(* Logix 5000 project; controller QW361 vendor 1 type 14 code 107 rev 32.11; software revision 32.00; part 16 of 20 *)

        [2374].log_data[1].valid := 1, [2374].log_data[2].valid := 1, [2374].log_data[3].valid := 1, [2374].log_data[4].valid := 1, [2374].time.Year := 2022, [2374].time.Month := 5, [2374].time.Day := 2, [2374].time.Hour := 3, [2374].time.Minute := 24, [2374].time.Second := 59, [2374].time.DST_ON := 1, [2375].log_data[0].min := 1.0, [2375].log_data[0].max := 1.0, [2375].log_data[0].total := 300.0, [2375].log_data[0].time := 300.0, [2375].log_data[0].minminute := 25, [2375].log_data[0].maxminute := 25, [2375].log_data[0].valid := 1, [2375].log_data[1].valid := 1, [2375].log_data[2].valid := 1, [2375].log_data[3].valid := 1, [2375].log_data[4].valid := 1, [2375].time.Year := 2022, [2375].time.Month := 5, [2375].time.Day := 2, [2375].time.Hour := 3, [2375].time.Minute := 29, [2375].time.Second := 59, [2375].time.DST_ON := 1, [2376].log_data[0].min := 1.0, [2376].log_data[0].max := 1.0, [2376].log_data[0].total := 300.0, [2376].log_data[0].time := 300.0, [2376].log_data[0].minminute := 30, [2376].log_data[0].maxminute := 30, [2376].log_data[0].valid := 1, [2376].log_data[1].valid := 1, [2376].log_data[2].valid := 1, [2376].log_data[3].valid := 1, [2376].log_data[4].valid := 1, [2376].time.Year := 2022, [2376].time.Month := 5, [2376].time.Day := 2, [2376].time.Hour := 3, [2376].time.Minute := 34, [2376].time.Second := 59, [2376].time.DST_ON := 1, [2377].log_data[0].min := 1.0, [2377].log_data[0].max := 1.0, [2377].log_data[0].total := 300.0, [2377].log_data[0].time := 300.0, [2377].log_data[0].minminute := 35, [2377].log_data[0].maxminute := 35, [2377].log_data[0].valid := 1, [2377].log_data[1].valid := 1, [2377].log_data[2].valid := 1, [2377].log_data[3].valid := 1, [2377].log_data[4].valid := 1, [2377].time.Year := 2022, [2377].time.Month := 5,
        [2377].time.Day := 2, [2377].time.Hour := 3, [2377].time.Minute := 39, [2377].time.Second := 59, [2377].time.DST_ON := 1, [2378].log_data[0].min := 1.0, [2378].log_data[0].max := 1.0, [2378].log_data[0].total := 300.0, [2378].log_data[0].time := 300.0, [2378].log_data[0].minminute := 40, [2378].log_data[0].maxminute := 40, [2378].log_data[0].valid := 1, [2378].log_data[1].valid := 1, [2378].log_data[2].valid := 1, [2378].log_data[3].valid := 1, [2378].log_data[4].valid := 1, [2378].time.Year := 2022, [2378].time.Month := 5, [2378].time.Day := 2, [2378].time.Hour := 3, [2378].time.Minute := 44, [2378].time.Second := 59, [2378].time.DST_ON := 1, [2379].log_data[0].min := 1.0, [2379].log_data[0].max := 1.0, [2379].log_data[0].total := 300.0, [2379].log_data[0].time := 300.0, [2379].log_data[0].minminute := 45, [2379].log_data[0].maxminute := 45, [2379].log_data[0].valid := 1, [2379].log_data[1].valid := 1, [2379].log_data[2].valid := 1, [2379].log_data[3].valid := 1, [2379].log_data[4].valid := 1, [2379].time.Year := 2022, [2379].time.Month := 5, [2379].time.Day := 2, [2379].time.Hour := 3, [2379].time.Minute := 49, [2379].time.Second := 59, [2379].time.DST_ON := 1, [2380].log_data[0].min := 1.0, [2380].log_data[0].max := 1.0, [2380].log_data[0].total := 300.0, [2380].log_data[0].time := 300.0, [2380].log_data[0].minminute := 50, [2380].log_data[0].maxminute := 50, [2380].log_data[0].valid := 1, [2380].log_data[1].valid := 1, [2380].log_data[2].valid := 1, [2380].log_data[3].valid := 1, [2380].log_data[4].valid := 1, [2380].time.Year := 2022, [2380].time.Month := 5, [2380].time.Day := 2, [2380].time.Hour := 3, [2380].time.Minute := 54, [2380].time.Second := 59, [2380].time.DST_ON := 1, [2381].log_data[0].min := 1.0,
        [2381].log_data[0].max := 1.0, [2381].log_data[0].total := 300.0, [2381].log_data[0].time := 300.0, [2381].log_data[0].minminute := 55, [2381].log_data[0].maxminute := 55, [2381].log_data[0].valid := 1, [2381].log_data[1].valid := 1, [2381].log_data[2].valid := 1, [2381].log_data[3].valid := 1, [2381].log_data[4].valid := 1, [2381].time.Year := 2022, [2381].time.Month := 5, [2381].time.Day := 2, [2381].time.Hour := 3, [2381].time.Minute := 59, [2381].time.Second := 59, [2381].time.DST_ON := 1, [2382].log_data[0].min := 1.0, [2382].log_data[0].max := 1.0, [2382].log_data[0].total := 300.0, [2382].log_data[0].time := 300.0, [2382].log_data[0].valid := 1, [2382].log_data[1].valid := 1, [2382].log_data[2].valid := 1, [2382].log_data[3].valid := 1, [2382].log_data[4].valid := 1, [2382].time.Year := 2022, [2382].time.Month := 5, [2382].time.Day := 2, [2382].time.Hour := 4, [2382].time.Minute := 4, [2382].time.Second := 59, [2382].time.DST_ON := 1, [2383].log_data[0].min := 1.0, [2383].log_data[0].max := 1.0, [2383].log_data[0].total := 300.0, [2383].log_data[0].time := 300.0, [2383].log_data[0].minminute := 5, [2383].log_data[0].maxminute := 5, [2383].log_data[0].valid := 1, [2383].log_data[1].valid := 1, [2383].log_data[2].valid := 1, [2383].log_data[3].valid := 1, [2383].log_data[4].valid := 1, [2383].time.Year := 2022, [2383].time.Month := 5, [2383].time.Day := 2, [2383].time.Hour := 4, [2383].time.Minute := 9, [2383].time.Second := 59, [2383].time.DST_ON := 1, [2384].log_data[0].min := 1.0, [2384].log_data[0].max := 1.0, [2384].log_data[0].total := 300.0, [2384].log_data[0].time := 300.0, [2384].log_data[0].minminute := 10, [2384].log_data[0].maxminute := 10, [2384].log_data[0].valid := 1, [2384].log_data[1].valid := 1, [2384].log_data[2].valid := 1,
        [2384].log_data[3].valid := 1, [2384].log_data[4].valid := 1, [2384].time.Year := 2022, [2384].time.Month := 5, [2384].time.Day := 2, [2384].time.Hour := 4, [2384].time.Minute := 14, [2384].time.Second := 59, [2384].time.DST_ON := 1, [2385].log_data[0].min := 1.0, [2385].log_data[0].max := 1.0, [2385].log_data[0].total := 300.0, [2385].log_data[0].time := 300.0, [2385].log_data[0].minminute := 15, [2385].log_data[0].maxminute := 15, [2385].log_data[0].valid := 1, [2385].log_data[1].valid := 1, [2385].log_data[2].valid := 1, [2385].log_data[3].valid := 1, [2385].log_data[4].valid := 1, [2385].time.Year := 2022, [2385].time.Month := 5, [2385].time.Day := 2, [2385].time.Hour := 4, [2385].time.Minute := 19, [2385].time.Second := 59, [2385].time.DST_ON := 1, [2386].log_data[0].min := 1.0, [2386].log_data[0].max := 1.0, [2386].log_data[0].total := 300.0, [2386].log_data[0].time := 300.0, [2386].log_data[0].minminute := 20, [2386].log_data[0].maxminute := 20, [2386].log_data[0].valid := 1, [2386].log_data[1].valid := 1, [2386].log_data[2].valid := 1, [2386].log_data[3].valid := 1, [2386].log_data[4].valid := 1, [2386].time.Year := 2022, [2386].time.Month := 5, [2386].time.Day := 2, [2386].time.Hour := 4, [2386].time.Minute := 24, [2386].time.Second := 59, [2386].time.DST_ON := 1, [2387].log_data[0].min := 1.0, [2387].log_data[0].max := 1.0, [2387].log_data[0].total := 300.0, [2387].log_data[0].time := 300.0, [2387].log_data[0].minminute := 25, [2387].log_data[0].maxminute := 25, [2387].log_data[0].valid := 1, [2387].log_data[1].valid := 1, [2387].log_data[2].valid := 1, [2387].log_data[3].valid := 1, [2387].log_data[4].valid := 1, [2387].time.Year := 2022, [2387].time.Month := 5, [2387].time.Day := 2, [2387].time.Hour := 4,
        [2387].time.Minute := 29, [2387].time.Second := 59, [2387].time.DST_ON := 1, [2388].log_data[0].min := 1.0, [2388].log_data[0].max := 1.0, [2388].log_data[0].total := 300.0, [2388].log_data[0].time := 300.0, [2388].log_data[0].minminute := 30, [2388].log_data[0].maxminute := 30, [2388].log_data[0].valid := 1, [2388].log_data[1].valid := 1, [2388].log_data[2].valid := 1, [2388].log_data[3].valid := 1, [2388].log_data[4].valid := 1, [2388].time.Year := 2022, [2388].time.Month := 5, [2388].time.Day := 2, [2388].time.Hour := 4, [2388].time.Minute := 34, [2388].time.Second := 59, [2388].time.DST_ON := 1, [2389].log_data[0].min := 1.0, [2389].log_data[0].max := 1.0, [2389].log_data[0].total := 300.0, [2389].log_data[0].time := 300.0, [2389].log_data[0].minminute := 35, [2389].log_data[0].maxminute := 35, [2389].log_data[0].valid := 1, [2389].log_data[1].valid := 1, [2389].log_data[2].valid := 1, [2389].log_data[3].valid := 1, [2389].log_data[4].valid := 1, [2389].time.Year := 2022, [2389].time.Month := 5, [2389].time.Day := 2, [2389].time.Hour := 4, [2389].time.Minute := 39, [2389].time.Second := 59, [2389].time.DST_ON := 1, [2390].log_data[0].min := 1.0, [2390].log_data[0].max := 1.0, [2390].log_data[0].total := 300.0, [2390].log_data[0].time := 300.0, [2390].log_data[0].minminute := 40, [2390].log_data[0].maxminute := 40, [2390].log_data[0].valid := 1, [2390].log_data[1].valid := 1, [2390].log_data[2].valid := 1, [2390].log_data[3].valid := 1, [2390].log_data[4].valid := 1, [2390].time.Year := 2022, [2390].time.Month := 5, [2390].time.Day := 2, [2390].time.Hour := 4, [2390].time.Minute := 44, [2390].time.Second := 59, [2390].time.DST_ON := 1, [2391].log_data[0].min := 1.0, [2391].log_data[0].max := 1.0, [2391].log_data[0].total := 300.0,
        [2391].log_data[0].time := 300.0, [2391].log_data[0].minminute := 45, [2391].log_data[0].maxminute := 45, [2391].log_data[0].valid := 1, [2391].log_data[1].valid := 1, [2391].log_data[2].valid := 1, [2391].log_data[3].valid := 1, [2391].log_data[4].valid := 1, [2391].time.Year := 2022, [2391].time.Month := 5, [2391].time.Day := 2, [2391].time.Hour := 4, [2391].time.Minute := 49, [2391].time.Second := 59, [2391].time.DST_ON := 1, [2392].log_data[0].min := 1.0, [2392].log_data[0].max := 1.0, [2392].log_data[0].total := 300.0, [2392].log_data[0].time := 300.0, [2392].log_data[0].minminute := 50, [2392].log_data[0].maxminute := 50, [2392].log_data[0].valid := 1, [2392].log_data[1].valid := 1, [2392].log_data[2].valid := 1, [2392].log_data[3].valid := 1, [2392].log_data[4].valid := 1, [2392].time.Year := 2022, [2392].time.Month := 5, [2392].time.Day := 2, [2392].time.Hour := 4, [2392].time.Minute := 54, [2392].time.Second := 59, [2392].time.DST_ON := 1, [2393].log_data[0].min := 1.0, [2393].log_data[0].max := 1.0, [2393].log_data[0].total := 300.0, [2393].log_data[0].time := 300.0, [2393].log_data[0].minminute := 55, [2393].log_data[0].maxminute := 55, [2393].log_data[0].valid := 1, [2393].log_data[1].valid := 1, [2393].log_data[2].valid := 1, [2393].log_data[3].valid := 1, [2393].log_data[4].valid := 1, [2393].time.Year := 2022, [2393].time.Month := 5, [2393].time.Day := 2, [2393].time.Hour := 4, [2393].time.Minute := 59, [2393].time.Second := 59, [2393].time.DST_ON := 1, [2394].log_data[0].min := 1.0, [2394].log_data[0].max := 1.0, [2394].log_data[0].total := 300.0, [2394].log_data[0].time := 300.0, [2394].log_data[0].valid := 1, [2394].log_data[1].valid := 1, [2394].log_data[2].valid := 1, [2394].log_data[3].valid := 1, [2394].log_data[4].valid := 1,
        [2394].time.Year := 2022, [2394].time.Month := 5, [2394].time.Day := 2, [2394].time.Hour := 5, [2394].time.Minute := 4, [2394].time.Second := 59, [2394].time.DST_ON := 1, [2395].log_data[0].min := 1.0, [2395].log_data[0].max := 1.0, [2395].log_data[0].total := 300.0, [2395].log_data[0].time := 300.0, [2395].log_data[0].minminute := 5, [2395].log_data[0].maxminute := 5, [2395].log_data[0].valid := 1, [2395].log_data[1].valid := 1, [2395].log_data[2].valid := 1, [2395].log_data[3].valid := 1, [2395].log_data[4].valid := 1, [2395].time.Year := 2022, [2395].time.Month := 5, [2395].time.Day := 2, [2395].time.Hour := 5, [2395].time.Minute := 9, [2395].time.Second := 59, [2395].time.DST_ON := 1, [2396].log_data[0].min := 1.0, [2396].log_data[0].max := 1.0, [2396].log_data[0].total := 300.0, [2396].log_data[0].time := 300.0, [2396].log_data[0].minminute := 10, [2396].log_data[0].maxminute := 10, [2396].log_data[0].valid := 1, [2396].log_data[1].valid := 1, [2396].log_data[2].valid := 1, [2396].log_data[3].valid := 1, [2396].log_data[4].valid := 1, [2396].time.Year := 2022, [2396].time.Month := 5, [2396].time.Day := 2, [2396].time.Hour := 5, [2396].time.Minute := 14, [2396].time.Second := 59, [2396].time.DST_ON := 1, [2397].log_data[0].min := 1.0, [2397].log_data[0].max := 1.0, [2397].log_data[0].total := 300.0, [2397].log_data[0].time := 300.0, [2397].log_data[0].minminute := 15, [2397].log_data[0].maxminute := 15, [2397].log_data[0].valid := 1, [2397].log_data[1].valid := 1, [2397].log_data[2].valid := 1, [2397].log_data[3].valid := 1, [2397].log_data[4].valid := 1, [2397].time.Year := 2022, [2397].time.Month := 5, [2397].time.Day := 2, [2397].time.Hour := 5, [2397].time.Minute := 19, [2397].time.Second := 59,
        [2397].time.DST_ON := 1, [2398].log_data[0].min := 1.0, [2398].log_data[0].max := 1.0, [2398].log_data[0].total := 300.0, [2398].log_data[0].time := 300.0, [2398].log_data[0].minminute := 20, [2398].log_data[0].maxminute := 20, [2398].log_data[0].valid := 1, [2398].log_data[1].valid := 1, [2398].log_data[2].valid := 1, [2398].log_data[3].valid := 1, [2398].log_data[4].valid := 1, [2398].time.Year := 2022, [2398].time.Month := 5, [2398].time.Day := 2, [2398].time.Hour := 5, [2398].time.Minute := 24, [2398].time.Second := 59, [2398].time.DST_ON := 1, [2399].log_data[0].min := 1.0, [2399].log_data[0].max := 1.0, [2399].log_data[0].total := 300.0, [2399].log_data[0].time := 300.0, [2399].log_data[0].minminute := 25, [2399].log_data[0].maxminute := 25, [2399].log_data[0].valid := 1, [2399].log_data[1].valid := 1, [2399].log_data[2].valid := 1, [2399].log_data[3].valid := 1, [2399].log_data[4].valid := 1, [2399].time.Year := 2022, [2399].time.Month := 5, [2399].time.Day := 2, [2399].time.Hour := 5, [2399].time.Minute := 29, [2399].time.Second := 59, [2399].time.DST_ON := 1);
   report5_row_qty : DINT := 2400;
   report_data : LogRecord[200] := ([0].log_data[0].min := 1.0, [0].log_data[0].max := 1.0, [0].log_data[0].total := 3600.5, [0].log_data[0].time := 3600.5, [0].log_data[0].valid := 1, [0].log_data[1].max := 1.0, [0].log_data[1].total := 503.5, [0].log_data[1].time := 3600.5, [0].log_data[1].maxminute := 28, [0].log_data[1].valid := 1, [0].log_data[2].time := 3600.5, [0].log_data[2].valid := 1, [0].log_data[3].time := 3600.5, [0].log_data[3].valid := 1, [0].log_data[4].min := 0.48749998, [0].log_data[4].max := 1.0068749, [0].log_data[4].total := 2840.4355, [0].log_data[4].time := 3600.5, [0].log_data[4].minminute := 37, [0].log_data[4].maxminute := 28, [0].log_data[4].valid := 1, [0].log_data[5].max := 7.1225, [0].log_data[5].total := 3526.124, [0].log_data[5].time := 3600.5, [0].log_data[5].maxminute := 30, [0].log_data[5].valid := 1, [0].log_data[6].valid := 1, [0].log_data[7].valid := 1, [0].log_data[8].valid := 1, [0].log_data[9].valid := 1, [0].log_data[10].valid := 1, [0].log_data[11].valid := 1, [0].log_data[12].valid := 1, [0].log_data[13].valid := 1, [0].log_data[14].valid := 1, [0].log_data[15].valid := 1, [0].log_data[16].valid := 1, [0].log_data[17].valid := 1, [0].log_data[18].valid := 1, [0].log_data[19].valid := 1, [0].time.Year := 2022, [0].time.Month := 4, [0].time.Day := 26, [0].time.Hour := 17, [0].time.Minute := 59, [0].time.Second := 59, [0].time.DST_ON := 1, [1].log_data[0].min := 1.0, [1].log_data[0].max := 1.0, [1].log_data[0].total := 3600.0, [1].log_data[0].time := 3600.0, [1].log_data[0].valid := 1, [1].log_data[1].time := 3600.0, [1].log_data[1].valid := 1, [1].log_data[2].max := 1.0, [1].log_data[2].total := 76.25, [1].log_data[2].time := 3600.0, [1].log_data[2].maxminute := 58, [1].log_data[2].valid := 1, [1].log_data[3].time := 3600.0,
        [1].log_data[3].valid := 1, [1].log_data[4].min := 0.6875, [1].log_data[4].max := 1.0068749, [1].log_data[4].total := 3210.5554, [1].log_data[4].time := 3600.0, [1].log_data[4].maxminute := 58, [1].log_data[4].valid := 1, [1].log_data[5].max := 7.2575, [1].log_data[5].total := 496.56125, [1].log_data[5].time := 3600.0, [1].log_data[5].maxminute := 59, [1].log_data[5].valid := 1, [1].log_data[6].valid := 1, [1].log_data[7].valid := 1, [1].log_data[8].valid := 1, [1].log_data[9].valid := 1, [1].log_data[10].valid := 1, [1].log_data[11].valid := 1, [1].log_data[12].valid := 1, [1].log_data[13].valid := 1, [1].log_data[14].valid := 1, [1].log_data[15].valid := 1, [1].log_data[16].valid := 1, [1].log_data[17].valid := 1, [1].log_data[18].valid := 1, [1].log_data[19].valid := 1, [1].time.Year := 2022, [1].time.Month := 4, [1].time.Day := 26, [1].time.Hour := 18, [1].time.Minute := 59, [1].time.Second := 59, [1].time.DST_ON := 1, [2].log_data[0].min := 1.0, [2].log_data[0].max := 1.0, [2].log_data[0].total := 3600.0, [2].log_data[0].time := 3600.0, [2].log_data[0].valid := 1, [2].log_data[1].time := 3600.0, [2].log_data[1].valid := 1, [2].log_data[2].max := 1.0, [2].log_data[2].total := 412.25, [2].log_data[2].time := 3600.0, [2].log_data[2].minminute := 6, [2].log_data[2].valid := 1, [2].log_data[3].time := 3600.0, [2].log_data[3].valid := 1, [2].log_data[4].min := 0.48812497, [2].log_data[4].max := 0.964375, [2].log_data[4].total := 2452.1655, [2].log_data[4].time := 3600.0, [2].log_data[4].minminute := 7, [2].log_data[4].valid := 1, [2].log_data[5].max := 7.25375, [2].log_data[5].total := 2977.3484, [2].log_data[5].time := 3600.0, [2].log_data[5].minminute := 7, [2].log_data[5].valid := 1, [2].log_data[6].valid := 1, [2].log_data[7].valid := 1,
        [2].log_data[8].valid := 1, [2].log_data[9].valid := 1, [2].log_data[10].valid := 1, [2].log_data[11].valid := 1, [2].log_data[12].valid := 1, [2].log_data[13].valid := 1, [2].log_data[14].valid := 1, [2].log_data[15].valid := 1, [2].log_data[16].valid := 1, [2].log_data[17].valid := 1, [2].log_data[18].valid := 1, [2].log_data[19].valid := 1, [2].time.Year := 2022, [2].time.Month := 4, [2].time.Day := 26, [2].time.Hour := 19, [2].time.Minute := 59, [2].time.Second := 59, [2].time.DST_ON := 1, [3].log_data[0].min := 1.0, [3].log_data[0].max := 1.0, [3].log_data[0].total := 3599.999, [3].log_data[0].time := 3599.999, [3].log_data[0].valid := 1, [3].log_data[1].max := 1.0, [3].log_data[1].total := 509.0, [3].log_data[1].time := 3599.999, [3].log_data[1].maxminute := 26, [3].log_data[1].valid := 1, [3].log_data[2].time := 3599.999, [3].log_data[2].valid := 1, [3].log_data[3].time := 3599.999, [3].log_data[3].valid := 1, [3].log_data[4].min := 0.48812497, [3].log_data[4].max := 1.00625, [3].log_data[4].total := 2816.658, [3].log_data[4].time := 3599.999, [3].log_data[4].minminute := 35, [3].log_data[4].maxminute := 26, [3].log_data[4].valid := 1, [3].log_data[5].max := 7.14375, [3].log_data[5].total := 3567.0015, [3].log_data[5].time := 3599.999, [3].log_data[5].maxminute := 27, [3].log_data[5].valid := 1, [3].log_data[6].valid := 1, [3].log_data[7].valid := 1, [3].log_data[8].valid := 1, [3].log_data[9].valid := 1, [3].log_data[10].valid := 1, [3].log_data[11].valid := 1, [3].log_data[12].valid := 1, [3].log_data[13].valid := 1, [3].log_data[14].valid := 1, [3].log_data[15].valid := 1, [3].log_data[16].valid := 1, [3].log_data[17].valid := 1, [3].log_data[18].valid := 1, [3].log_data[19].valid := 1, [3].time.Year := 2022,
        [3].time.Month := 4, [3].time.Day := 26, [3].time.Hour := 20, [3].time.Minute := 59, [3].time.Second := 59, [3].time.DST_ON := 1, [4].log_data[0].min := 1.0, [4].log_data[0].max := 1.0, [4].log_data[0].total := 3600.0, [4].log_data[0].time := 3600.0, [4].log_data[0].valid := 1, [4].log_data[1].time := 3600.0, [4].log_data[1].valid := 1, [4].log_data[2].max := 1.0, [4].log_data[2].total := 520.5, [4].log_data[2].time := 3600.0, [4].log_data[2].maxminute := 36, [4].log_data[2].valid := 1, [4].log_data[3].time := 3600.0, [4].log_data[3].valid := 1, [4].log_data[4].min := 0.48812497, [4].log_data[4].max := 1.0068749, [4].log_data[4].total := 2907.509, [4].log_data[4].time := 3600.0, [4].log_data[4].minminute := 45, [4].log_data[4].maxminute := 36, [4].log_data[4].valid := 1, [4].log_data[5].max := 7.22875, [4].log_data[5].total := 3690.3572, [4].log_data[5].time := 3600.0, [4].log_data[5].maxminute := 37, [4].log_data[5].valid := 1, [4].log_data[6].valid := 1, [4].log_data[7].valid := 1, [4].log_data[8].valid := 1, [4].log_data[9].valid := 1, [4].log_data[10].valid := 1, [4].log_data[11].valid := 1, [4].log_data[12].valid := 1, [4].log_data[13].valid := 1, [4].log_data[14].valid := 1, [4].log_data[15].valid := 1, [4].log_data[16].valid := 1, [4].log_data[17].valid := 1, [4].log_data[18].valid := 1, [4].log_data[19].valid := 1, [4].time.Year := 2022, [4].time.Month := 4, [4].time.Day := 26, [4].time.Hour := 21, [4].time.Minute := 59, [4].time.Second := 59, [4].time.DST_ON := 1, [5].log_data[0].min := 1.0, [5].log_data[0].max := 1.0, [5].log_data[0].total := 3600.0, [5].log_data[0].time := 3600.0, [5].log_data[0].valid := 1, [5].log_data[1].max := 1.0, [5].log_data[1].total := 509.5,
        [5].log_data[1].time := 3600.0, [5].log_data[1].maxminute := 46, [5].log_data[1].valid := 1, [5].log_data[2].time := 3600.0, [5].log_data[2].valid := 1, [5].log_data[3].time := 3600.0, [5].log_data[3].valid := 1, [5].log_data[4].min := 0.48812497, [5].log_data[4].max := 1.0068749, [5].log_data[4].total := 3018.5044, [5].log_data[4].time := 3600.0, [5].log_data[4].minminute := 55, [5].log_data[4].maxminute := 47, [5].log_data[4].valid := 1, [5].log_data[5].max := 7.133749, [5].log_data[5].total := 3577.1904, [5].log_data[5].time := 3600.0, [5].log_data[5].maxminute := 48, [5].log_data[5].valid := 1, [5].log_data[6].valid := 1, [5].log_data[7].valid := 1, [5].log_data[8].valid := 1, [5].log_data[9].valid := 1, [5].log_data[10].valid := 1, [5].log_data[11].valid := 1, [5].log_data[12].valid := 1, [5].log_data[13].valid := 1, [5].log_data[14].valid := 1, [5].log_data[15].valid := 1, [5].log_data[16].valid := 1, [5].log_data[17].valid := 1, [5].log_data[18].valid := 1, [5].log_data[19].valid := 1, [5].time.Year := 2022, [5].time.Month := 4, [5].time.Day := 26, [5].time.Hour := 22, [5].time.Minute := 59, [5].time.Second := 59, [5].time.DST_ON := 1, [6].log_data[0].min := 1.0, [6].log_data[0].max := 1.0, [6].log_data[0].total := 3599.999, [6].log_data[0].time := 3599.999, [6].log_data[0].valid := 1, [6].log_data[1].time := 3599.999, [6].log_data[1].valid := 1, [6].log_data[2].time := 3599.999, [6].log_data[2].valid := 1, [6].log_data[3].time := 3599.999, [6].log_data[3].valid := 1, [6].log_data[4].min := 0.534375, [6].log_data[4].max := 0.94875, [6].log_data[4].total := 2817.2761, [6].log_data[4].time := 3599.999, [6].log_data[4].maxminute := 58, [6].log_data[4].valid := 1, [6].log_data[5].max := 0.0012500001, [6].log_data[5].total := 1.5889835, [6].log_data[5].time := 3599.999,
        [6].log_data[5].valid := 1, [6].log_data[6].valid := 1, [6].log_data[7].valid := 1, [6].log_data[8].valid := 1, [6].log_data[9].valid := 1, [6].log_data[10].valid := 1, [6].log_data[11].valid := 1, [6].log_data[12].valid := 1, [6].log_data[13].valid := 1, [6].log_data[14].valid := 1, [6].log_data[15].valid := 1, [6].log_data[16].valid := 1, [6].log_data[17].valid := 1, [6].log_data[18].valid := 1, [6].log_data[19].valid := 1, [6].time.Year := 2022, [6].time.Month := 4, [6].time.Day := 26, [6].time.Hour := 23, [6].time.Minute := 59, [6].time.Second := 59, [6].time.DST_ON := 1, [7].log_data[0].min := 1.0, [7].log_data[0].max := 1.0, [7].log_data[0].total := 3600.0, [7].log_data[0].time := 3600.0, [7].log_data[0].valid := 1, [7].log_data[1].time := 3600.0, [7].log_data[1].valid := 1, [7].log_data[2].max := 1.0, [7].log_data[2].total := 486.0, [7].log_data[2].time := 3600.0, [7].log_data[2].maxminute := 19, [7].log_data[2].valid := 1, [7].log_data[3].time := 3600.0, [7].log_data[3].valid := 1, [7].log_data[4].min := 0.48812497, [7].log_data[4].max := 1.005625, [7].log_data[4].total := 2770.1392, [7].log_data[4].time := 3600.0, [7].log_data[4].minminute := 27, [7].log_data[4].maxminute := 19, [7].log_data[4].valid := 1, [7].log_data[5].max := 7.2337503, [7].log_data[5].total := 3454.3674, [7].log_data[5].time := 3600.0, [7].log_data[5].maxminute := 20, [7].log_data[5].valid := 1, [7].log_data[6].valid := 1, [7].log_data[7].valid := 1, [7].log_data[8].valid := 1, [7].log_data[9].valid := 1, [7].log_data[10].valid := 1, [7].log_data[11].valid := 1, [7].log_data[12].valid := 1, [7].log_data[13].valid := 1, [7].log_data[14].valid := 1, [7].log_data[15].valid := 1, [7].log_data[16].valid := 1, [7].log_data[17].valid := 1,
        [7].log_data[18].valid := 1, [7].log_data[19].valid := 1, [7].time.Year := 2022, [7].time.Month := 4, [7].time.Day := 27, [7].time.Minute := 59, [7].time.Second := 59, [7].time.DST_ON := 1, [8].log_data[0].min := 1.0, [8].log_data[0].max := 1.0, [8].log_data[0].total := 3600.0, [8].log_data[0].time := 3600.0, [8].log_data[0].valid := 1, [8].log_data[1].time := 3600.0, [8].log_data[1].valid := 1, [8].log_data[2].time := 3600.0, [8].log_data[2].valid := 1, [8].log_data[3].time := 3600.0, [8].log_data[3].valid := 1, [8].log_data[4].min := 0.79499996, [8].log_data[4].max := 0.98, [8].log_data[4].total := 3282.462, [8].log_data[4].time := 3600.0, [8].log_data[4].maxminute := 57, [8].log_data[4].valid := 1, [8].log_data[5].max := 0.0012500001, [8].log_data[5].total := 2.463077, [8].log_data[5].time := 3600.0, [8].log_data[5].valid := 1, [8].log_data[6].valid := 1, [8].log_data[7].valid := 1, [8].log_data[8].valid := 1, [8].log_data[9].valid := 1, [8].log_data[10].valid := 1, [8].log_data[11].valid := 1, [8].log_data[12].valid := 1, [8].log_data[13].valid := 1, [8].log_data[14].valid := 1, [8].log_data[15].valid := 1, [8].log_data[16].valid := 1, [8].log_data[17].valid := 1, [8].log_data[18].valid := 1, [8].log_data[19].valid := 1, [8].time.Year := 2022, [8].time.Month := 4, [8].time.Day := 27, [8].time.Hour := 1, [8].time.Minute := 59, [8].time.Second := 59, [8].time.DST_ON := 1, [9].log_data[0].min := 1.0, [9].log_data[0].max := 1.0, [9].log_data[0].total := 3600.0, [9].log_data[0].time := 3600.0, [9].log_data[0].valid := 1, [9].log_data[1].max := 1.0, [9].log_data[1].total := 472.0, [9].log_data[1].time := 3600.0, [9].log_data[1].maxminute := 27, [9].log_data[1].valid := 1,
        [9].log_data[2].time := 3600.0, [9].log_data[2].valid := 1, [9].log_data[3].time := 3600.0, [9].log_data[3].valid := 1, [9].log_data[4].min := 0.48812497, [9].log_data[4].max := 1.005, [9].log_data[4].total := 2770.1748, [9].log_data[4].time := 3600.0, [9].log_data[4].minminute := 35, [9].log_data[4].maxminute := 27, [9].log_data[4].valid := 1, [9].log_data[5].max := 7.1512504, [9].log_data[5].total := 3321.189, [9].log_data[5].time := 3600.0, [9].log_data[5].maxminute := 28, [9].log_data[5].valid := 1, [9].log_data[6].valid := 1, [9].log_data[7].valid := 1, [9].log_data[8].valid := 1, [9].log_data[9].valid := 1, [9].log_data[10].valid := 1, [9].log_data[11].valid := 1, [9].log_data[12].valid := 1, [9].log_data[13].valid := 1, [9].log_data[14].valid := 1, [9].log_data[15].valid := 1, [9].log_data[16].valid := 1, [9].log_data[17].valid := 1, [9].log_data[18].valid := 1, [9].log_data[19].valid := 1, [9].time.Year := 2022, [9].time.Month := 4, [9].time.Day := 27, [9].time.Hour := 2, [9].time.Minute := 59, [9].time.Second := 59, [9].time.DST_ON := 1, [10].log_data[0].min := 1.0, [10].log_data[0].max := 1.0, [10].log_data[0].total := 3599.999, [10].log_data[0].time := 3599.999, [10].log_data[0].valid := 1, [10].log_data[1].time := 3599.999, [10].log_data[1].valid := 1, [10].log_data[2].time := 3599.999, [10].log_data[2].valid := 1, [10].log_data[3].time := 3599.999, [10].log_data[3].valid := 1, [10].log_data[4].min := 0.55, [10].log_data[4].max := 0.68875, [10].log_data[4].total := 2235.2305, [10].log_data[4].time := 3599.999, [10].log_data[4].maxminute := 56, [10].log_data[4].valid := 1, [10].log_data[5].max := 0.0012500001, [10].log_data[5].total := 3.2619953, [10].log_data[5].time := 3599.999, [10].log_data[5].valid := 1, [10].log_data[6].valid := 1, [10].log_data[7].valid := 1,
        [10].log_data[8].valid := 1, [10].log_data[9].valid := 1, [10].log_data[10].valid := 1, [10].log_data[11].valid := 1, [10].log_data[12].valid := 1, [10].log_data[13].valid := 1, [10].log_data[14].valid := 1, [10].log_data[15].valid := 1, [10].log_data[16].valid := 1, [10].log_data[17].valid := 1, [10].log_data[18].valid := 1, [10].log_data[19].valid := 1, [10].time.Year := 2022, [10].time.Month := 4, [10].time.Day := 27, [10].time.Hour := 3, [10].time.Minute := 59, [10].time.Second := 59, [10].time.DST_ON := 1, [11].log_data[0].min := 1.0, [11].log_data[0].max := 1.0, [11].log_data[0].total := 3600.0, [11].log_data[0].time := 3600.0, [11].log_data[0].valid := 1, [11].log_data[1].time := 3600.0, [11].log_data[1].valid := 1, [11].log_data[2].time := 3600.0, [11].log_data[2].valid := 1, [11].log_data[3].time := 3600.0, [11].log_data[3].valid := 1, [11].log_data[4].min := 0.68812495, [11].log_data[4].max := 0.8106251, [11].log_data[4].total := 2699.7146, [11].log_data[4].time := 3600.0, [11].log_data[4].maxminute := 56, [11].log_data[4].valid := 1, [11].log_data[5].max := 0.0012500001, [11].log_data[5].total := 3.3301373, [11].log_data[5].time := 3600.0, [11].log_data[5].valid := 1, [11].log_data[6].valid := 1, [11].log_data[7].valid := 1, [11].log_data[8].valid := 1, [11].log_data[9].valid := 1, [11].log_data[10].valid := 1, [11].log_data[11].valid := 1, [11].log_data[12].valid := 1, [11].log_data[13].valid := 1, [11].log_data[14].valid := 1, [11].log_data[15].valid := 1, [11].log_data[16].valid := 1, [11].log_data[17].valid := 1, [11].log_data[18].valid := 1, [11].log_data[19].valid := 1, [11].time.Year := 2022, [11].time.Month := 4, [11].time.Day := 27, [11].time.Hour := 4, [11].time.Minute := 59, [11].time.Second := 59,
        [11].time.DST_ON := 1, [12].log_data[0].min := 1.0, [12].log_data[0].max := 1.0, [12].log_data[0].total := 3599.999, [12].log_data[0].time := 3599.999, [12].log_data[0].valid := 1, [12].log_data[1].time := 3599.999, [12].log_data[1].valid := 1, [12].log_data[2].time := 3599.999, [12].log_data[2].valid := 1, [12].log_data[3].time := 3599.999, [12].log_data[3].valid := 1, [12].log_data[4].min := 0.81, [12].log_data[4].max := 0.888125, [12].log_data[4].total := 3082.9211, [12].log_data[4].time := 3599.999, [12].log_data[4].maxminute := 49, [12].log_data[4].valid := 1, [12].log_data[5].max := 0.0025000002, [12].log_data[5].total := 3.538617, [12].log_data[5].time := 3599.999, [12].log_data[5].maxminute := 4, [12].log_data[5].valid := 1, [12].log_data[6].valid := 1, [12].log_data[7].valid := 1, [12].log_data[8].valid := 1, [12].log_data[9].valid := 1, [12].log_data[10].valid := 1, [12].log_data[11].valid := 1, [12].log_data[12].valid := 1, [12].log_data[13].valid := 1, [12].log_data[14].valid := 1, [12].log_data[15].valid := 1, [12].log_data[16].valid := 1, [12].log_data[17].valid := 1, [12].log_data[18].valid := 1, [12].log_data[19].valid := 1, [12].time.Year := 2022, [12].time.Month := 4, [12].time.Day := 27, [12].time.Hour := 5, [12].time.Minute := 59, [12].time.Second := 59, [12].time.DST_ON := 1, [13].log_data[0].min := 1.0, [13].log_data[0].max := 1.0, [13].log_data[0].total := 3600.0, [13].log_data[0].time := 3600.0, [13].log_data[0].valid := 1, [13].log_data[1].time := 3600.0, [13].log_data[1].valid := 1, [13].log_data[2].time := 3600.0, [13].log_data[2].valid := 1, [13].log_data[3].time := 3600.0, [13].log_data[3].valid := 1, [13].log_data[4].min := 0.8875, [13].log_data[4].max := 0.934375, [13].log_data[4].total := 3295.0835, [13].log_data[4].time := 3600.0, [13].log_data[4].maxminute := 45,
        [13].log_data[4].valid := 1, [13].log_data[5].max := 0.0025000002, [13].log_data[5].total := 3.5189261, [13].log_data[5].time := 3600.0, [13].log_data[5].maxminute := 8, [13].log_data[5].valid := 1, [13].log_data[6].valid := 1, [13].log_data[7].valid := 1, [13].log_data[8].valid := 1, [13].log_data[9].valid := 1, [13].log_data[10].valid := 1, [13].log_data[11].valid := 1, [13].log_data[12].valid := 1, [13].log_data[13].valid := 1, [13].log_data[14].valid := 1, [13].log_data[15].valid := 1, [13].log_data[16].valid := 1, [13].log_data[17].valid := 1, [13].log_data[18].valid := 1, [13].log_data[19].valid := 1, [13].time.Year := 2022, [13].time.Month := 4, [13].time.Day := 27, [13].time.Hour := 6, [13].time.Minute := 59, [13].time.Second := 59, [13].time.DST_ON := 1, [14].log_data[0].min := 1.0, [14].log_data[0].max := 1.0, [14].log_data[0].total := 3600.0, [14].log_data[0].time := 3600.0, [14].log_data[0].valid := 1, [14].log_data[1].time := 3600.0, [14].log_data[1].valid := 1, [14].log_data[2].time := 3600.0, [14].log_data[2].valid := 1, [14].log_data[3].time := 3600.0, [14].log_data[3].valid := 1, [14].log_data[4].min := 0.93375, [14].log_data[4].max := 0.99687505, [14].log_data[4].total := 3460.6003, [14].log_data[4].time := 3600.0, [14].log_data[4].maxminute := 59, [14].log_data[4].valid := 1, [14].log_data[5].max := 0.0012500001, [14].log_data[5].total := 3.5773764, [14].log_data[5].time := 3600.0, [14].log_data[5].valid := 1, [14].log_data[6].valid := 1, [14].log_data[7].valid := 1, [14].log_data[8].valid := 1, [14].log_data[9].valid := 1, [14].log_data[10].valid := 1, [14].log_data[11].valid := 1, [14].log_data[12].valid := 1, [14].log_data[13].valid := 1, [14].log_data[14].valid := 1, [14].log_data[15].valid := 1, [14].log_data[16].valid := 1, [14].log_data[17].valid := 1,
        [14].log_data[18].valid := 1, [14].log_data[19].valid := 1, [14].time.Year := 2022, [14].time.Month := 4, [14].time.Day := 27, [14].time.Hour := 7, [14].time.Minute := 59, [14].time.Second := 59, [14].time.DST_ON := 1, [15].log_data[0].min := 1.0, [15].log_data[0].max := 1.0, [15].log_data[0].total := 3600.0, [15].log_data[0].time := 3600.0, [15].log_data[0].valid := 1, [15].log_data[1].time := 3600.0, [15].log_data[1].valid := 1, [15].log_data[2].max := 1.0, [15].log_data[2].total := 475.5, [15].log_data[2].time := 3600.0, [15].log_data[2].valid := 1, [15].log_data[3].time := 3600.0, [15].log_data[3].valid := 1, [15].log_data[4].min := 0.48812497, [15].log_data[4].max := 1.0068749, [15].log_data[4].total := 2464.974, [15].log_data[4].time := 3600.0, [15].log_data[4].minminute := 8, [15].log_data[4].valid := 1, [15].log_data[5].max := 7.34375, [15].log_data[5].total := 3421.07, [15].log_data[5].time := 3600.0, [15].log_data[5].maxminute := 1, [15].log_data[5].valid := 1, [15].log_data[6].valid := 1, [15].log_data[7].valid := 1, [15].log_data[8].valid := 1, [15].log_data[9].valid := 1, [15].log_data[10].valid := 1, [15].log_data[11].valid := 1, [15].log_data[12].valid := 1, [15].log_data[13].valid := 1, [15].log_data[14].valid := 1, [15].log_data[15].valid := 1, [15].log_data[16].valid := 1, [15].log_data[17].valid := 1, [15].log_data[18].valid := 1, [15].log_data[19].valid := 1, [15].time.Year := 2022, [15].time.Month := 4, [15].time.Day := 27, [15].time.Hour := 8, [15].time.Minute := 59, [15].time.Second := 59, [15].time.DST_ON := 1, [16].log_data[0].min := 1.0, [16].log_data[0].max := 1.0, [16].log_data[0].total := 3600.0, [16].log_data[0].time := 3600.0, [16].log_data[0].valid := 1, [16].log_data[1].max := 1.0,
        [16].log_data[1].total := 500.5, [16].log_data[1].time := 3600.0, [16].log_data[1].maxminute := 35, [16].log_data[1].valid := 1, [16].log_data[2].time := 3600.0, [16].log_data[2].valid := 1, [16].log_data[3].time := 3600.0, [16].log_data[3].valid := 1, [16].log_data[4].min := 0.48812497, [16].log_data[4].max := 1.0074999, [16].log_data[4].total := 2912.9893, [16].log_data[4].time := 3600.0, [16].log_data[4].minminute := 43, [16].log_data[4].maxminute := 35, [16].log_data[4].valid := 1, [16].log_data[5].max := 7.1550007, [16].log_data[5].total := 3524.6697, [16].log_data[5].time := 3600.0, [16].log_data[5].maxminute := 37, [16].log_data[5].valid := 1, [16].log_data[6].valid := 1, [16].log_data[7].valid := 1, [16].log_data[8].valid := 1, [16].log_data[9].valid := 1, [16].log_data[10].valid := 1, [16].log_data[11].valid := 1, [16].log_data[12].valid := 1, [16].log_data[13].valid := 1, [16].log_data[14].valid := 1, [16].log_data[15].valid := 1, [16].log_data[16].valid := 1, [16].log_data[17].valid := 1, [16].log_data[18].valid := 1, [16].log_data[19].valid := 1, [16].time.Year := 2022, [16].time.Month := 4, [16].time.Day := 27, [16].time.Hour := 9, [16].time.Minute := 59, [16].time.Second := 59, [16].time.DST_ON := 1, [17].log_data[0].min := 1.0, [17].log_data[0].max := 1.0, [17].log_data[0].total := 3600.0, [17].log_data[0].time := 3600.0, [17].log_data[0].valid := 1, [17].log_data[1].time := 3600.0, [17].log_data[1].valid := 1, [17].log_data[2].time := 3600.0, [17].log_data[2].valid := 1, [17].log_data[3].time := 3600.0, [17].log_data[3].valid := 1, [17].log_data[4].min := 0.6112499, [17].log_data[4].max := 0.98, [17].log_data[4].total := 2937.459, [17].log_data[4].time := 3600.0, [17].log_data[4].maxminute := 58, [17].log_data[4].valid := 1, [17].log_data[5].max := 0.0012500001, [17].log_data[5].total := 1.1221869,
        [17].log_data[5].time := 3600.0, [17].log_data[5].valid := 1, [17].log_data[6].valid := 1, [17].log_data[7].valid := 1, [17].log_data[8].valid := 1, [17].log_data[9].valid := 1, [17].log_data[10].valid := 1, [17].log_data[11].valid := 1, [17].log_data[12].valid := 1, [17].log_data[13].valid := 1, [17].log_data[14].valid := 1, [17].log_data[15].valid := 1, [17].log_data[16].valid := 1, [17].log_data[17].valid := 1, [17].log_data[18].valid := 1, [17].log_data[19].valid := 1, [17].time.Year := 2022, [17].time.Month := 4, [17].time.Day := 27, [17].time.Hour := 10, [17].time.Minute := 59, [17].time.Second := 59, [17].time.DST_ON := 1, [18].log_data[0].min := 1.0, [18].log_data[0].max := 1.0, [18].log_data[0].total := 3600.0, [18].log_data[0].time := 3600.0, [18].log_data[0].valid := 1, [18].log_data[1].max := 1.0, [18].log_data[1].total := 138.0, [18].log_data[1].time := 3600.0, [18].log_data[1].maxminute := 21, [18].log_data[1].valid := 1, [18].log_data[2].max := 1.0, [18].log_data[2].total := 621.5, [18].log_data[2].time := 3600.0, [18].log_data[2].maxminute := 7, [18].log_data[2].valid := 1, [18].log_data[3].time := 3600.0, [18].log_data[3].valid := 1, [18].log_data[4].min := 0.32000002, [18].log_data[4].max := 1.0074999, [18].log_data[4].total := 2164.0217, [18].log_data[4].time := 3600.0, [18].log_data[4].minminute := 23, [18].log_data[4].maxminute := 7, [18].log_data[4].valid := 1, [18].log_data[5].max := 8.615, [18].log_data[5].total := 4677.1943, [18].log_data[5].time := 3600.0, [18].log_data[5].maxminute := 22, [18].log_data[5].valid := 1, [18].log_data[6].valid := 1, [18].log_data[7].valid := 1, [18].log_data[8].valid := 1, [18].log_data[9].valid := 1, [18].log_data[10].valid := 1, [18].log_data[11].valid := 1, [18].log_data[12].valid := 1, [18].log_data[13].valid := 1,
        [18].log_data[14].valid := 1, [18].log_data[15].valid := 1, [18].log_data[16].valid := 1, [18].log_data[17].valid := 1, [18].log_data[18].valid := 1, [18].log_data[19].valid := 1, [18].time.Year := 2022, [18].time.Month := 4, [18].time.Day := 27, [18].time.Hour := 11, [18].time.Minute := 59, [18].time.Second := 59, [18].time.DST_ON := 1, [19].log_data[0].min := 1.0, [19].log_data[0].max := 1.0, [19].log_data[0].total := 3600.0, [19].log_data[0].time := 3600.0, [19].log_data[0].valid := 1, [19].log_data[1].time := 3600.0, [19].log_data[1].valid := 1, [19].log_data[2].time := 3600.0, [19].log_data[2].valid := 1, [19].log_data[3].time := 3600.0, [19].log_data[3].valid := 1, [19].log_data[4].min := 0.6725, [19].log_data[4].max := 0.95, [19].log_data[4].total := 3046.559, [19].log_data[4].time := 3600.0, [19].log_data[4].maxminute := 59, [19].log_data[4].valid := 1, [19].log_data[5].max := 0.0025000002, [19].log_data[5].total := 0.9918947, [19].log_data[5].time := 3600.0, [19].log_data[5].maxminute := 7, [19].log_data[5].valid := 1, [19].log_data[6].valid := 1, [19].log_data[7].valid := 1, [19].log_data[8].valid := 1, [19].log_data[9].valid := 1, [19].log_data[10].valid := 1, [19].log_data[11].valid := 1, [19].log_data[12].valid := 1, [19].log_data[13].valid := 1, [19].log_data[14].valid := 1, [19].log_data[15].valid := 1, [19].log_data[16].valid := 1, [19].log_data[17].valid := 1, [19].log_data[18].valid := 1, [19].log_data[19].valid := 1, [19].time.Year := 2022, [19].time.Month := 4, [19].time.Day := 27, [19].time.Hour := 12, [19].time.Minute := 59, [19].time.Second := 59, [19].time.DST_ON := 1, [20].log_data[0].min := 1.0, [20].log_data[0].max := 1.0, [20].log_data[0].total := 3600.0, [20].log_data[0].time := 3600.0,
        [20].log_data[0].valid := 1, [20].log_data[1].max := 1.0, [20].log_data[1].total := 483.0, [20].log_data[1].time := 3600.0, [20].log_data[1].maxminute := 20, [20].log_data[1].valid := 1, [20].log_data[2].time := 3600.0, [20].log_data[2].valid := 1, [20].log_data[3].time := 3600.0, [20].log_data[3].valid := 1, [20].log_data[4].min := 0.48812497, [20].log_data[4].max := 1.0068749, [20].log_data[4].total := 2650.4507, [20].log_data[4].time := 3600.0, [20].log_data[4].minminute := 29, [20].log_data[4].maxminute := 20, [20].log_data[4].valid := 1, [20].log_data[5].max := 7.14375, [20].log_data[5].total := 3387.5083, [20].log_data[5].time := 3600.0, [20].log_data[5].maxminute := 21, [20].log_data[5].valid := 1, [20].log_data[6].valid := 1, [20].log_data[7].valid := 1, [20].log_data[8].valid := 1, [20].log_data[9].valid := 1, [20].log_data[10].valid := 1, [20].log_data[11].valid := 1, [20].log_data[12].valid := 1, [20].log_data[13].valid := 1, [20].log_data[14].valid := 1, [20].log_data[15].valid := 1, [20].log_data[16].valid := 1, [20].log_data[17].valid := 1, [20].log_data[18].valid := 1, [20].log_data[19].valid := 1, [20].time.Year := 2022, [20].time.Month := 4, [20].time.Day := 27, [20].time.Hour := 13, [20].time.Minute := 59, [20].time.Second := 59, [20].time.DST_ON := 1, [21].log_data[0].min := 1.0, [21].log_data[0].max := 1.0, [21].log_data[0].total := 3600.0, [21].log_data[0].time := 3600.0, [21].log_data[0].valid := 1, [21].log_data[1].time := 3600.0, [21].log_data[1].valid := 1, [21].log_data[2].time := 3600.0, [21].log_data[2].valid := 1, [21].log_data[3].time := 3600.0, [21].log_data[3].valid := 1, [21].log_data[4].min := 0.62624997, [21].log_data[4].max := 0.85687506, [21].log_data[4].total := 2670.7908, [21].log_data[4].time := 3600.0, [21].log_data[4].maxminute := 56, [21].log_data[4].valid := 1,
        [21].log_data[5].max := 0.0012500001, [21].log_data[5].total := 0.13281257, [21].log_data[5].time := 3600.0, [21].log_data[5].valid := 1, [21].log_data[6].valid := 1, [21].log_data[7].valid := 1, [21].log_data[8].valid := 1, [21].log_data[9].valid := 1, [21].log_data[10].valid := 1, [21].log_data[11].valid := 1, [21].log_data[12].valid := 1, [21].log_data[13].valid := 1, [21].log_data[14].valid := 1, [21].log_data[15].valid := 1, [21].log_data[16].valid := 1, [21].log_data[17].valid := 1, [21].log_data[18].valid := 1, [21].log_data[19].valid := 1, [21].time.Year := 2022, [21].time.Month := 4, [21].time.Day := 27, [21].time.Hour := 14, [21].time.Minute := 59, [21].time.Second := 59, [21].time.DST_ON := 1, [22].log_data[0].min := 1.0, [22].log_data[0].max := 1.0, [22].log_data[0].total := 3599.999, [22].log_data[0].time := 3599.999, [22].log_data[0].valid := 1, [22].log_data[1].time := 3599.999, [22].log_data[1].valid := 1, [22].log_data[2].time := 3599.999, [22].log_data[2].valid := 1, [22].log_data[3].time := 3599.999, [22].log_data[3].valid := 1, [22].log_data[4].min := 0.85625, [22].log_data[4].max := 0.995, [22].log_data[4].total := 3357.9556, [22].log_data[4].time := 3599.999, [22].log_data[4].maxminute := 57, [22].log_data[4].valid := 1, [22].log_data[5].max := 0.0012500001, [22].log_data[5].total := 0.1203124, [22].log_data[5].time := 3599.999, [22].log_data[5].valid := 1, [22].log_data[6].valid := 1, [22].log_data[7].valid := 1, [22].log_data[8].valid := 1, [22].log_data[9].valid := 1, [22].log_data[10].valid := 1, [22].log_data[11].valid := 1, [22].log_data[12].valid := 1, [22].log_data[13].valid := 1, [22].log_data[14].valid := 1, [22].log_data[15].valid := 1, [22].log_data[16].valid := 1, [22].log_data[17].valid := 1, [22].log_data[18].valid := 1, [22].log_data[19].valid := 1,
        [22].time.Year := 2022, [22].time.Month := 4, [22].time.Day := 27, [22].time.Hour := 15, [22].time.Minute := 59, [22].time.Second := 59, [22].time.DST_ON := 1, [23].log_data[0].min := 1.0, [23].log_data[0].max := 1.0, [23].log_data[0].total := 3600.0, [23].log_data[0].time := 3600.0, [23].log_data[0].valid := 1, [23].log_data[1].time := 3600.0, [23].log_data[1].valid := 1, [23].log_data[2].max := 1.0, [23].log_data[2].total := 474.5, [23].log_data[2].time := 3600.0, [23].log_data[2].maxminute := 6, [23].log_data[2].valid := 1, [23].log_data[3].time := 3600.0, [23].log_data[3].valid := 1, [23].log_data[4].min := 0.48812497, [23].log_data[4].max := 1.003125, [23].log_data[4].total := 2454.8042, [23].log_data[4].time := 3600.0, [23].log_data[4].minminute := 14, [23].log_data[4].maxminute := 6, [23].log_data[4].valid := 1, [23].log_data[5].max := 7.28125, [23].log_data[5].total := 3389.3877, [23].log_data[5].time := 3600.0, [23].log_data[5].maxminute := 7, [23].log_data[5].valid := 1, [23].log_data[6].valid := 1, [23].log_data[7].valid := 1, [23].log_data[8].valid := 1, [23].log_data[9].valid := 1, [23].log_data[10].valid := 1, [23].log_data[11].valid := 1, [23].log_data[12].valid := 1, [23].log_data[13].valid := 1, [23].log_data[14].valid := 1, [23].log_data[15].valid := 1, [23].log_data[16].valid := 1, [23].log_data[17].valid := 1, [23].log_data[18].valid := 1, [23].log_data[19].valid := 1, [23].time.Year := 2022, [23].time.Month := 4, [23].time.Day := 27, [23].time.Hour := 16, [23].time.Minute := 59, [23].time.Second := 59, [23].time.DST_ON := 1, [24].log_data[0].min := 1.0, [24].log_data[0].max := 1.0, [24].log_data[0].total := 3599.999, [24].log_data[0].time := 3599.999, [24].log_data[0].valid := 1, [24].log_data[1].max := 1.0,
        [24].log_data[1].total := 441.75, [24].log_data[1].time := 3599.999, [24].log_data[1].maxminute := 52, [24].log_data[1].valid := 1, [24].log_data[2].time := 3599.999, [24].log_data[2].valid := 1, [24].log_data[3].time := 3599.999, [24].log_data[3].valid := 1, [24].log_data[4].min := 0.56875, [24].log_data[4].max := 1.0074999, [24].log_data[4].total := 3275.0847, [24].log_data[4].time := 3599.999, [24].log_data[4].minminute := 59, [24].log_data[4].maxminute := 52, [24].log_data[4].valid := 1, [24].log_data[5].max := 7.13125, [24].log_data[5].total := 3067.3916, [24].log_data[5].time := 3599.999, [24].log_data[5].maxminute := 53, [24].log_data[5].valid := 1, [24].log_data[6].valid := 1, [24].log_data[7].valid := 1, [24].log_data[8].valid := 1, [24].log_data[9].valid := 1, [24].log_data[10].valid := 1, [24].log_data[11].valid := 1, [24].log_data[12].valid := 1, [24].log_data[13].valid := 1, [24].log_data[14].valid := 1, [24].log_data[15].valid := 1, [24].log_data[16].valid := 1, [24].log_data[17].valid := 1, [24].log_data[18].valid := 1, [24].log_data[19].valid := 1, [24].time.Year := 2022, [24].time.Month := 4, [24].time.Day := 27, [24].time.Hour := 17, [24].time.Minute := 59, [24].time.Second := 59, [24].time.DST_ON := 1, [25].log_data[0].min := 1.0, [25].log_data[0].max := 1.0, [25].log_data[0].total := 3600.0, [25].log_data[0].time := 3600.0, [25].log_data[0].valid := 1, [25].log_data[1].max := 1.0, [25].log_data[1].total := 50.25, [25].log_data[1].time := 3600.0, [25].log_data[1].valid := 1, [25].log_data[2].time := 3600.0, [25].log_data[2].valid := 1, [25].log_data[3].time := 3600.0, [25].log_data[3].valid := 1, [25].log_data[4].min := 0.48812497, [25].log_data[4].max := 0.934375, [25].log_data[4].total := 2602.4575, [25].log_data[4].time := 3600.0, [25].log_data[4].minminute := 1, [25].log_data[4].maxminute := 59,
        [25].log_data[4].valid := 1, [25].log_data[5].max := 6.9674993, [25].log_data[5].total := 386.91257, [25].log_data[5].time := 3600.0, [25].log_data[5].minminute := 1, [25].log_data[5].valid := 1, [25].log_data[6].valid := 1, [25].log_data[7].valid := 1, [25].log_data[8].valid := 1, [25].log_data[9].valid := 1, [25].log_data[10].valid := 1, [25].log_data[11].valid := 1, [25].log_data[12].valid := 1, [25].log_data[13].valid := 1, [25].log_data[14].valid := 1, [25].log_data[15].valid := 1, [25].log_data[16].valid := 1, [25].log_data[17].valid := 1, [25].log_data[18].valid := 1, [25].log_data[19].valid := 1, [25].time.Year := 2022, [25].time.Month := 4, [25].time.Day := 27, [25].time.Hour := 18, [25].time.Minute := 59, [25].time.Second := 59, [25].time.DST_ON := 1, [26].log_data[0].min := 1.0, [26].log_data[0].max := 1.0, [26].log_data[0].total := 3599.999, [26].log_data[0].time := 3599.999, [26].log_data[0].valid := 1, [26].log_data[1].time := 3599.999, [26].log_data[1].valid := 1, [26].log_data[2].max := 1.0, [26].log_data[2].total := 488.5, [26].log_data[2].time := 3599.999, [26].log_data[2].maxminute := 20, [26].log_data[2].valid := 1, [26].log_data[3].time := 3599.999, [26].log_data[3].valid := 1, [26].log_data[4].min := 0.48812497, [26].log_data[4].max := 1.0074999, [26].log_data[4].total := 2716.5222, [26].log_data[4].time := 3599.999, [26].log_data[4].minminute := 28, [26].log_data[4].maxminute := 20, [26].log_data[4].valid := 1, [26].log_data[5].max := 7.3125, [26].log_data[5].total := 3509.2307, [26].log_data[5].time := 3599.999, [26].log_data[5].maxminute := 21, [26].log_data[5].valid := 1, [26].log_data[6].valid := 1, [26].log_data[7].valid := 1, [26].log_data[8].valid := 1, [26].log_data[9].valid := 1, [26].log_data[10].valid := 1, [26].log_data[11].valid := 1, [26].log_data[12].valid := 1,
        [26].log_data[13].valid := 1, [26].log_data[14].valid := 1, [26].log_data[15].valid := 1, [26].log_data[16].valid := 1, [26].log_data[17].valid := 1, [26].log_data[18].valid := 1, [26].log_data[19].valid := 1, [26].time.Year := 2022, [26].time.Month := 4, [26].time.Day := 27, [26].time.Hour := 19, [26].time.Minute := 59, [26].time.Second := 59, [26].time.DST_ON := 1, [27].log_data[0].min := 1.0, [27].log_data[0].max := 1.0, [27].log_data[0].total := 3599.999, [27].log_data[0].time := 3599.999, [27].log_data[0].valid := 1, [27].log_data[1].max := 1.0, [27].log_data[1].total := 442.25, [27].log_data[1].time := 3599.999, [27].log_data[1].maxminute := 52, [27].log_data[1].valid := 1, [27].log_data[2].time := 3599.999, [27].log_data[2].valid := 1, [27].log_data[3].time := 3599.999, [27].log_data[3].valid := 1, [27].log_data[4].min := 0.60437495, [27].log_data[4].max := 1.0074999, [27].log_data[4].total := 3165.9084, [27].log_data[4].time := 3599.999, [27].log_data[4].minminute := 59, [27].log_data[4].maxminute := 52, [27].log_data[4].valid := 1, [27].log_data[5].max := 7.13625, [27].log_data[5].total := 3072.2383, [27].log_data[5].time := 3599.999, [27].log_data[5].maxminute := 53, [27].log_data[5].valid := 1, [27].log_data[6].valid := 1, [27].log_data[7].valid := 1, [27].log_data[8].valid := 1, [27].log_data[9].valid := 1, [27].log_data[10].valid := 1, [27].log_data[11].valid := 1, [27].log_data[12].valid := 1, [27].log_data[13].valid := 1, [27].log_data[14].valid := 1, [27].log_data[15].valid := 1, [27].log_data[16].valid := 1, [27].log_data[17].valid := 1, [27].log_data[18].valid := 1, [27].log_data[19].valid := 1, [27].time.Year := 2022, [27].time.Month := 4, [27].time.Day := 27, [27].time.Hour := 20, [27].time.Minute := 59, [27].time.Second := 59,
        [27].time.DST_ON := 1, [28].log_data[0].min := 1.0, [28].log_data[0].max := 1.0, [28].log_data[0].total := 3600.0, [28].log_data[0].time := 3600.0, [28].log_data[0].valid := 1, [28].log_data[1].max := 1.0, [28].log_data[1].total := 81.75, [28].log_data[1].time := 3600.0, [28].log_data[1].minminute := 1, [28].log_data[1].valid := 1, [28].log_data[2].max := 1.0, [28].log_data[2].total := 349.25, [28].log_data[2].time := 3600.0, [28].log_data[2].maxminute := 54, [28].log_data[2].valid := 1, [28].log_data[3].time := 3600.0, [28].log_data[3].valid := 1, [28].log_data[4].min := 0.48812497, [28].log_data[4].max := 1.0074999, [28].log_data[4].total := 2863.1797, [28].log_data[4].time := 3600.0, [28].log_data[4].minminute := 1, [28].log_data[4].maxminute := 54, [28].log_data[4].valid := 1, [28].log_data[5].max := 7.23125, [28].log_data[5].total := 3050.0334, [28].log_data[5].time := 3600.0, [28].log_data[5].minminute := 1, [28].log_data[5].maxminute := 55, [28].log_data[5].valid := 1, [28].log_data[6].valid := 1, [28].log_data[7].valid := 1, [28].log_data[8].valid := 1, [28].log_data[9].valid := 1, [28].log_data[10].valid := 1, [28].log_data[11].valid := 1, [28].log_data[12].valid := 1, [28].log_data[13].valid := 1, [28].log_data[14].valid := 1, [28].log_data[15].valid := 1, [28].log_data[16].valid := 1, [28].log_data[17].valid := 1, [28].log_data[18].valid := 1, [28].log_data[19].valid := 1, [28].time.Year := 2022, [28].time.Month := 4, [28].time.Day := 27, [28].time.Hour := 21, [28].time.Minute := 59, [28].time.Second := 59, [28].time.DST_ON := 1, [29].log_data[0].min := 1.0, [29].log_data[0].max := 1.0, [29].log_data[0].total := 3600.0, [29].log_data[0].time := 3600.0, [29].log_data[0].valid := 1, [29].log_data[1].time := 3600.0, [29].log_data[1].valid := 1, [29].log_data[2].max := 1.0,
        [29].log_data[2].total := 158.25, [29].log_data[2].time := 3600.0, [29].log_data[2].minminute := 2, [29].log_data[2].valid := 1, [29].log_data[3].time := 3600.0, [29].log_data[3].valid := 1, [29].log_data[4].min := 0.48812497, [29].log_data[4].max := 0.95875, [29].log_data[4].total := 2747.6846, [29].log_data[4].time := 3600.0, [29].log_data[4].minminute := 2, [29].log_data[4].maxminute := 59, [29].log_data[4].valid := 1, [29].log_data[5].max := 7.11875, [29].log_data[5].total := 1156.4518, [29].log_data[5].time := 3600.0, [29].log_data[5].minminute := 2, [29].log_data[5].valid := 1, [29].log_data[6].valid := 1, [29].log_data[7].valid := 1, [29].log_data[8].valid := 1, [29].log_data[9].valid := 1, [29].log_data[10].valid := 1, [29].log_data[11].valid := 1, [29].log_data[12].valid := 1, [29].log_data[13].valid := 1, [29].log_data[14].valid := 1, [29].log_data[15].valid := 1, [29].log_data[16].valid := 1, [29].log_data[17].valid := 1, [29].log_data[18].valid := 1, [29].log_data[19].valid := 1, [29].time.Year := 2022, [29].time.Month := 4, [29].time.Day := 27, [29].time.Hour := 22, [29].time.Minute := 59, [29].time.Second := 59, [29].time.DST_ON := 1, [30].log_data[0].min := 1.0, [30].log_data[0].max := 1.0, [30].log_data[0].total := 3599.999, [30].log_data[0].time := 3599.999, [30].log_data[0].valid := 1, [30].log_data[1].max := 1.0, [30].log_data[1].total := 479.499, [30].log_data[1].time := 3599.999, [30].log_data[1].maxminute := 17, [30].log_data[1].valid := 1, [30].log_data[2].time := 3599.999, [30].log_data[2].valid := 1, [30].log_data[3].time := 3599.999, [30].log_data[3].valid := 1, [30].log_data[4].min := 0.48812497, [30].log_data[4].max := 1.004375, [30].log_data[4].total := 2604.554, [30].log_data[4].time := 3599.999, [30].log_data[4].minminute := 25, [30].log_data[4].maxminute := 17, [30].log_data[4].valid := 1,
        [30].log_data[5].max := 7.2375, [30].log_data[5].total := 3412.6675, [30].log_data[5].time := 3599.999, [30].log_data[5].maxminute := 19, [30].log_data[5].valid := 1, [30].log_data[6].valid := 1, [30].log_data[7].valid := 1, [30].log_data[8].valid := 1, [30].log_data[9].valid := 1, [30].log_data[10].valid := 1, [30].log_data[11].valid := 1, [30].log_data[12].valid := 1, [30].log_data[13].valid := 1, [30].log_data[14].valid := 1, [30].log_data[15].valid := 1, [30].log_data[16].valid := 1, [30].log_data[17].valid := 1, [30].log_data[18].valid := 1, [30].log_data[19].valid := 1, [30].time.Year := 2022, [30].time.Month := 4, [30].time.Day := 27, [30].time.Hour := 23, [30].time.Minute := 59, [30].time.Second := 59, [30].time.DST_ON := 1, [31].log_data[0].min := 1.0, [31].log_data[0].max := 1.0, [31].log_data[0].total := 3600.0, [31].log_data[0].time := 3600.0, [31].log_data[0].valid := 1, [31].log_data[1].time := 3600.0, [31].log_data[1].valid := 1, [31].log_data[2].time := 3600.0, [31].log_data[2].valid := 1, [31].log_data[3].time := 3600.0, [31].log_data[3].valid := 1, [31].log_data[4].min := 0.6575, [31].log_data[4].max := 0.90312505, [31].log_data[4].total := 2891.3281, [31].log_data[4].time := 3600.0, [31].log_data[4].maxminute := 54, [31].log_data[4].valid := 1, [31].log_data[5].max := 0.0012500001, [31].log_data[5].total := 2.5802884, [31].log_data[5].time := 3600.0, [31].log_data[5].valid := 1, [31].log_data[6].valid := 1, [31].log_data[7].valid := 1, [31].log_data[8].valid := 1, [31].log_data[9].valid := 1, [31].log_data[10].valid := 1, [31].log_data[11].valid := 1, [31].log_data[12].valid := 1, [31].log_data[13].valid := 1, [31].log_data[14].valid := 1, [31].log_data[15].valid := 1, [31].log_data[16].valid := 1, [31].log_data[17].valid := 1, [31].log_data[18].valid := 1,
        [31].log_data[19].valid := 1, [31].time.Year := 2022, [31].time.Month := 4, [31].time.Day := 28, [31].time.Minute := 59, [31].time.Second := 59, [31].time.DST_ON := 1, [32].log_data[0].min := 1.0, [32].log_data[0].max := 1.0, [32].log_data[0].total := 3600.0, [32].log_data[0].time := 3600.0, [32].log_data[0].valid := 1, [32].log_data[1].time := 3600.0, [32].log_data[1].valid := 1, [32].log_data[2].max := 1.0, [32].log_data[2].total := 489.0, [32].log_data[2].time := 3600.0, [32].log_data[2].maxminute := 36, [32].log_data[2].valid := 1, [32].log_data[3].time := 3600.0, [32].log_data[3].valid := 1, [32].log_data[4].min := 0.48812497, [32].log_data[4].max := 1.0068749, [32].log_data[4].total := 2975.8533, [32].log_data[4].time := 3600.0, [32].log_data[4].minminute := 45, [32].log_data[4].maxminute := 36, [32].log_data[4].valid := 1, [32].log_data[5].max := 7.23625, [32].log_data[5].total := 3475.8203, [32].log_data[5].time := 3600.0, [32].log_data[5].maxminute := 38, [32].log_data[5].valid := 1, [32].log_data[6].valid := 1, [32].log_data[7].valid := 1, [32].log_data[8].valid := 1, [32].log_data[9].valid := 1, [32].log_data[10].valid := 1, [32].log_data[11].valid := 1, [32].log_data[12].valid := 1, [32].log_data[13].valid := 1, [32].log_data[14].valid := 1, [32].log_data[15].valid := 1, [32].log_data[16].valid := 1, [32].log_data[17].valid := 1, [32].log_data[18].valid := 1, [32].log_data[19].valid := 1, [32].time.Year := 2022, [32].time.Month := 4, [32].time.Day := 28, [32].time.Hour := 1, [32].time.Minute := 59, [32].time.Second := 59, [32].time.DST_ON := 1, [33].log_data[0].min := 1.0, [33].log_data[0].max := 1.0, [33].log_data[0].total := 3600.0, [33].log_data[0].time := 3600.0, [33].log_data[0].valid := 1, [33].log_data[1].time := 3600.0,
        [33].log_data[1].valid := 1, [33].log_data[2].time := 3600.0, [33].log_data[2].valid := 1, [33].log_data[3].time := 3600.0, [33].log_data[3].valid := 1, [33].log_data[4].min := 0.580625, [33].log_data[4].max := 0.81125, [33].log_data[4].total := 2532.1038, [33].log_data[4].time := 3600.0, [33].log_data[4].maxminute := 59, [33].log_data[4].valid := 1, [33].log_data[5].max := 0.0012500001, [33].log_data[5].total := 3.5376804, [33].log_data[5].time := 3600.0, [33].log_data[5].valid := 1, [33].log_data[6].valid := 1, [33].log_data[7].valid := 1, [33].log_data[8].valid := 1, [33].log_data[9].valid := 1, [33].log_data[10].valid := 1, [33].log_data[11].valid := 1, [33].log_data[12].valid := 1, [33].log_data[13].valid := 1, [33].log_data[14].valid := 1, [33].log_data[15].valid := 1, [33].log_data[16].valid := 1, [33].log_data[17].valid := 1, [33].log_data[18].valid := 1, [33].log_data[19].valid := 1, [33].time.Year := 2022, [33].time.Month := 4, [33].time.Day := 28, [33].time.Hour := 2, [33].time.Minute := 59, [33].time.Second := 59, [33].time.DST_ON := 1, [34].log_data[0].min := 1.0, [34].log_data[0].max := 1.0, [34].log_data[0].total := 3599.999, [34].log_data[0].time := 3599.999, [34].log_data[0].valid := 1, [34].log_data[1].time := 3599.999, [34].log_data[1].valid := 1, [34].log_data[2].time := 3599.999, [34].log_data[2].valid := 1, [34].log_data[3].time := 3599.999, [34].log_data[3].valid := 1, [34].log_data[4].min := 0.8106251, [34].log_data[4].max := 0.888125, [34].log_data[4].total := 3085.281, [34].log_data[4].time := 3599.999, [34].log_data[4].maxminute := 46, [34].log_data[4].valid := 1, [34].log_data[5].max := 0.0012500001, [34].log_data[5].total := 3.9368267, [34].log_data[5].time := 3599.999, [34].log_data[5].valid := 1, [34].log_data[6].valid := 1, [34].log_data[7].valid := 1, [34].log_data[8].valid := 1,
        [34].log_data[9].valid := 1, [34].log_data[10].valid := 1, [34].log_data[11].valid := 1, [34].log_data[12].valid := 1, [34].log_data[13].valid := 1, [34].log_data[14].valid := 1, [34].log_data[15].valid := 1, [34].log_data[16].valid := 1, [34].log_data[17].valid := 1, [34].log_data[18].valid := 1, [34].log_data[19].valid := 1, [34].time.Year := 2022, [34].time.Month := 4, [34].time.Day := 28, [34].time.Hour := 3, [34].time.Minute := 59, [34].time.Second := 59, [34].time.DST_ON := 1, [35].log_data[0].min := 1.0, [35].log_data[0].max := 1.0, [35].log_data[0].total := 3600.0, [35].log_data[0].time := 3600.0, [35].log_data[0].valid := 1, [35].log_data[1].time := 3600.0, [35].log_data[1].valid := 1, [35].log_data[2].time := 3600.0, [35].log_data[2].valid := 1, [35].log_data[3].time := 3600.0, [35].log_data[3].valid := 1, [35].log_data[4].min := 0.888125, [35].log_data[4].max := 0.965625, [35].log_data[4].total := 3308.7012, [35].log_data[4].time := 3600.0, [35].log_data[4].maxminute := 59, [35].log_data[4].valid := 1, [35].log_data[5].max := 0.0025000002, [35].log_data[5].total := 4.0730386, [35].log_data[5].time := 3600.0, [35].log_data[5].maxminute := 20, [35].log_data[5].valid := 1, [35].log_data[6].valid := 1, [35].log_data[7].valid := 1, [35].log_data[8].valid := 1, [35].log_data[9].valid := 1, [35].log_data[10].valid := 1, [35].log_data[11].valid := 1, [35].log_data[12].valid := 1, [35].log_data[13].valid := 1, [35].log_data[14].valid := 1, [35].log_data[15].valid := 1, [35].log_data[16].valid := 1, [35].log_data[17].valid := 1, [35].log_data[18].valid := 1, [35].log_data[19].valid := 1, [35].time.Year := 2022, [35].time.Month := 4, [35].time.Day := 28, [35].time.Hour := 4, [35].time.Minute := 59, [35].time.Second := 59,
        [35].time.DST_ON := 1, [36].log_data[0].min := 1.0, [36].log_data[0].max := 1.0, [36].log_data[0].total := 3600.0, [36].log_data[0].time := 3600.0, [36].log_data[0].valid := 1, [36].log_data[1].max := 1.0, [36].log_data[1].total := 477.5, [36].log_data[1].time := 3600.0, [36].log_data[1].maxminute := 25, [36].log_data[1].valid := 1, [36].log_data[2].time := 3600.0, [36].log_data[2].valid := 1, [36].log_data[3].time := 3600.0, [36].log_data[3].valid := 1, [36].log_data[4].min := 0.48812497, [36].log_data[4].max := 1.005625, [36].log_data[4].total := 2704.658, [36].log_data[4].time := 3600.0, [36].log_data[4].minminute := 35, [36].log_data[4].maxminute := 25, [36].log_data[4].valid := 1, [36].log_data[5].max := 7.1650004, [36].log_data[5].total := 3355.2085, [36].log_data[5].time := 3600.0, [36].log_data[5].maxminute := 26, [36].log_data[5].valid := 1, [36].log_data[6].valid := 1, [36].log_data[7].valid := 1, [36].log_data[8].valid := 1, [36].log_data[9].valid := 1, [36].log_data[10].valid := 1, [36].log_data[11].valid := 1, [36].log_data[12].valid := 1, [36].log_data[13].valid := 1, [36].log_data[14].valid := 1, [36].log_data[15].valid := 1, [36].log_data[16].valid := 1, [36].log_data[17].valid := 1, [36].log_data[18].valid := 1, [36].log_data[19].valid := 1, [36].time.Year := 2022, [36].time.Month := 4, [36].time.Day := 28, [36].time.Hour := 5, [36].time.Minute := 59, [36].time.Second := 59, [36].time.DST_ON := 1, [37].log_data[0].min := 1.0, [37].log_data[0].max := 1.0, [37].log_data[0].total := 3599.999, [37].log_data[0].time := 3599.999, [37].log_data[0].valid := 1, [37].log_data[1].time := 3599.999, [37].log_data[1].valid := 1, [37].log_data[2].time := 3599.999, [37].log_data[2].valid := 1, [37].log_data[3].time := 3599.999, [37].log_data[3].valid := 1, [37].log_data[4].min := 0.55062497,
        [37].log_data[4].max := 0.64312506, [37].log_data[4].total := 2128.7969, [37].log_data[4].time := 3599.999, [37].log_data[4].maxminute := 59, [37].log_data[4].valid := 1, [37].log_data[5].max := 0.0025000002, [37].log_data[5].total := 4.26763, [37].log_data[5].time := 3599.999, [37].log_data[5].maxminute := 3, [37].log_data[5].valid := 1, [37].log_data[6].valid := 1, [37].log_data[7].valid := 1, [37].log_data[8].valid := 1, [37].log_data[9].valid := 1, [37].log_data[10].valid := 1, [37].log_data[11].valid := 1, [37].log_data[12].valid := 1, [37].log_data[13].valid := 1, [37].log_data[14].valid := 1, [37].log_data[15].valid := 1, [37].log_data[16].valid := 1, [37].log_data[17].valid := 1, [37].log_data[18].valid := 1, [37].log_data[19].valid := 1, [37].time.Year := 2022, [37].time.Month := 4, [37].time.Day := 28, [37].time.Hour := 6, [37].time.Minute := 59, [37].time.Second := 59, [37].time.DST_ON := 1, [38].log_data[0].min := 1.0, [38].log_data[0].max := 1.0, [38].log_data[0].total := 3600.0, [38].log_data[0].time := 3600.0, [38].log_data[0].valid := 1, [38].log_data[1].time := 3600.0, [38].log_data[1].valid := 1, [38].log_data[2].time := 3600.0, [38].log_data[2].valid := 1, [38].log_data[3].time := 3600.0, [38].log_data[3].valid := 1, [38].log_data[4].min := 0.6425, [38].log_data[4].max := 0.87312496, [38].log_data[4].total := 2658.2312, [38].log_data[4].time := 3600.0, [38].log_data[4].minminute := 1, [38].log_data[4].maxminute := 59, [38].log_data[4].valid := 1, [38].log_data[5].max := 0.0025000002, [38].log_data[5].total := 3.7364728, [38].log_data[5].time := 3600.0, [38].log_data[5].valid := 1, [38].log_data[6].valid := 1, [38].log_data[7].valid := 1, [38].log_data[8].valid := 1, [38].log_data[9].valid := 1, [38].log_data[10].valid := 1, [38].log_data[11].valid := 1, [38].log_data[12].valid := 1,
        [38].log_data[13].valid := 1, [38].log_data[14].valid := 1, [38].log_data[15].valid := 1, [38].log_data[16].valid := 1, [38].log_data[17].valid := 1, [38].log_data[18].valid := 1, [38].log_data[19].valid := 1, [38].time.Year := 2022, [38].time.Month := 4, [38].time.Day := 28, [38].time.Hour := 7, [38].time.Minute := 59, [38].time.Second := 59, [38].time.DST_ON := 1, [39].log_data[0].min := 1.0, [39].log_data[0].max := 1.0, [39].log_data[0].total := 3600.0, [39].log_data[0].time := 3600.0, [39].log_data[0].valid := 1, [39].log_data[1].time := 3600.0, [39].log_data[1].valid := 1, [39].log_data[2].max := 1.0, [39].log_data[2].total := 521.0, [39].log_data[2].time := 3600.0, [39].log_data[2].maxminute := 23, [39].log_data[2].valid := 1, [39].log_data[3].time := 3600.0, [39].log_data[3].valid := 1, [39].log_data[4].min := 0.48874998, [39].log_data[4].max := 1.009375, [39].log_data[4].total := 2873.5457, [39].log_data[4].time := 3600.0, [39].log_data[4].minminute := 32, [39].log_data[4].maxminute := 24, [39].log_data[4].valid := 1, [39].log_data[5].max := 7.3287497, [39].log_data[5].total := 3750.9976, [39].log_data[5].time := 3600.0, [39].log_data[5].maxminute := 25, [39].log_data[5].valid := 1, [39].log_data[6].valid := 1, [39].log_data[7].valid := 1, [39].log_data[8].valid := 1, [39].log_data[9].valid := 1, [39].log_data[10].valid := 1, [39].log_data[11].valid := 1, [39].log_data[12].valid := 1, [39].log_data[13].valid := 1, [39].log_data[14].valid := 1, [39].log_data[15].valid := 1, [39].log_data[16].valid := 1, [39].log_data[17].valid := 1, [39].log_data[18].valid := 1, [39].log_data[19].valid := 1, [39].time.Year := 2022, [39].time.Month := 4, [39].time.Day := 28, [39].time.Hour := 8, [39].time.Minute := 59, [39].time.Second := 59,
        [39].time.DST_ON := 1, [40].log_data[0].min := 1.0, [40].log_data[0].max := 1.0, [40].log_data[0].total := 3600.0, [40].log_data[0].time := 3600.0, [40].log_data[0].valid := 1, [40].log_data[1].max := 1.0, [40].log_data[1].total := 495.0, [40].log_data[1].time := 3600.0, [40].log_data[1].maxminute := 33, [40].log_data[1].valid := 1, [40].log_data[2].time := 3600.0, [40].log_data[2].valid := 1, [40].log_data[3].time := 3600.0, [40].log_data[3].valid := 1, [40].log_data[4].min := 0.48812497, [40].log_data[4].max := 1.0081251, [40].log_data[4].total := 2897.89, [40].log_data[4].time := 3600.0, [40].log_data[4].minminute := 42, [40].log_data[4].maxminute := 33, [40].log_data[4].valid := 1, [40].log_data[5].max := 7.2237496, [40].log_data[5].total := 3508.4324, [40].log_data[5].time := 3600.0, [40].log_data[5].maxminute := 34, [40].log_data[5].valid := 1, [40].log_data[6].valid := 1, [40].log_data[7].valid := 1, [40].log_data[8].valid := 1, [40].log_data[9].valid := 1, [40].log_data[10].valid := 1, [40].log_data[11].valid := 1, [40].log_data[12].valid := 1, [40].log_data[13].valid := 1, [40].log_data[14].valid := 1, [40].log_data[15].valid := 1, [40].log_data[16].valid := 1, [40].log_data[17].valid := 1, [40].log_data[18].valid := 1, [40].log_data[19].valid := 1, [40].time.Year := 2022, [40].time.Month := 4, [40].time.Day := 28, [40].time.Hour := 9, [40].time.Minute := 59, [40].time.Second := 59, [40].time.DST_ON := 1, [41].log_data[0].min := 1.0, [41].log_data[0].max := 1.0, [41].log_data[0].total := 3599.999, [41].log_data[0].time := 3599.999, [41].log_data[0].valid := 1, [41].log_data[1].time := 3599.999, [41].log_data[1].valid := 1, [41].log_data[2].time := 3599.999, [41].log_data[2].valid := 1, [41].log_data[3].time := 3599.999, [41].log_data[3].valid := 1, [41].log_data[4].min := 0.62687504,
        [41].log_data[4].max := 0.9806249, [41].log_data[4].total := 2928.4136, [41].log_data[4].time := 3599.999, [41].log_data[4].maxminute := 58, [41].log_data[4].valid := 1, [41].log_data[5].max := 0.0012500001, [41].log_data[5].total := 0.09062493, [41].log_data[5].time := 3599.999, [41].log_data[5].valid := 1, [41].log_data[6].valid := 1, [41].log_data[7].valid := 1, [41].log_data[8].valid := 1, [41].log_data[9].valid := 1, [41].log_data[10].valid := 1, [41].log_data[11].valid := 1, [41].log_data[12].valid := 1, [41].log_data[13].valid := 1, [41].log_data[14].valid := 1, [41].log_data[15].valid := 1, [41].log_data[16].valid := 1, [41].log_data[17].valid := 1, [41].log_data[18].valid := 1, [41].log_data[19].valid := 1, [41].time.Year := 2022, [41].time.Month := 4, [41].time.Day := 28, [41].time.Hour := 10, [41].time.Minute := 59, [41].time.Second := 59, [41].time.DST_ON := 1, [42].log_data[0].min := 1.0, [42].log_data[0].max := 1.0, [42].log_data[0].total := 3600.0, [42].log_data[0].time := 3600.0, [42].log_data[0].valid := 1, [42].log_data[1].time := 3600.0, [42].log_data[1].valid := 1, [42].log_data[2].max := 1.0, [42].log_data[2].total := 494.5, [42].log_data[2].time := 3600.0, [42].log_data[2].maxminute := 5, [42].log_data[2].valid := 1, [42].log_data[3].time := 3600.0, [42].log_data[3].valid := 1, [42].log_data[4].min := 0.48812497, [42].log_data[4].max := 1.0074999, [42].log_data[4].total := 2550.2021, [42].log_data[4].time := 3600.0, [42].log_data[4].minminute := 14, [42].log_data[4].maxminute := 5, [42].log_data[4].valid := 1, [42].log_data[5].max := 7.25625, [42].log_data[5].total := 3513.8455, [42].log_data[5].time := 3600.0, [42].log_data[5].maxminute := 7, [42].log_data[5].valid := 1, [42].log_data[6].valid := 1, [42].log_data[7].valid := 1, [42].log_data[8].valid := 1, [42].log_data[9].valid := 1,
        [42].log_data[10].valid := 1, [42].log_data[11].valid := 1, [42].log_data[12].valid := 1, [42].log_data[13].valid := 1, [42].log_data[14].valid := 1, [42].log_data[15].valid := 1, [42].log_data[16].valid := 1, [42].log_data[17].valid := 1, [42].log_data[18].valid := 1, [42].log_data[19].valid := 1, [42].time.Year := 2022, [42].time.Month := 4, [42].time.Day := 28, [42].time.Hour := 11, [42].time.Minute := 59, [42].time.Second := 59, [42].time.DST_ON := 1, [43].log_data[0].min := 1.0, [43].log_data[0].max := 1.0, [43].log_data[0].total := 3600.0, [43].log_data[0].time := 3600.0, [43].log_data[0].valid := 1, [43].log_data[1].max := 1.0, [43].log_data[1].total := 388.25, [43].log_data[1].time := 3600.0, [43].log_data[1].maxminute := 53, [43].log_data[1].valid := 1, [43].log_data[2].time := 3600.0, [43].log_data[2].valid := 1, [43].log_data[3].time := 3600.0, [43].log_data[3].valid := 1, [43].log_data[4].min := 0.6375, [43].log_data[4].max := 1.0074999, [43].log_data[4].total := 3309.6946, [43].log_data[4].time := 3600.0, [43].log_data[4].minminute := 59, [43].log_data[4].maxminute := 53, [43].log_data[4].valid := 1, [43].log_data[5].max := 7.1825, [43].log_data[5].total := 2712.425, [43].log_data[5].time := 3600.0, [43].log_data[5].maxminute := 59, [43].log_data[5].valid := 1, [43].log_data[6].valid := 1, [43].log_data[7].valid := 1, [43].log_data[8].valid := 1, [43].log_data[9].valid := 1, [43].log_data[10].valid := 1, [43].log_data[11].valid := 1, [43].log_data[12].valid := 1, [43].log_data[13].valid := 1, [43].log_data[14].valid := 1, [43].log_data[15].valid := 1, [43].log_data[16].valid := 1, [43].log_data[17].valid := 1, [43].log_data[18].valid := 1, [43].log_data[19].valid := 1, [43].time.Year := 2022, [43].time.Month := 4, [43].time.Day := 28,
        [43].time.Hour := 12, [43].time.Minute := 59, [43].time.Second := 59, [43].time.DST_ON := 1, [44].log_data[0].min := 1.0, [44].log_data[0].max := 1.0, [44].log_data[0].total := 3600.0, [44].log_data[0].time := 3600.0, [44].log_data[0].valid := 1, [44].log_data[1].max := 1.0, [44].log_data[1].total := 95.25, [44].log_data[1].time := 3600.0, [44].log_data[1].minminute := 1, [44].log_data[1].valid := 1, [44].log_data[2].time := 3600.0, [44].log_data[2].valid := 1, [44].log_data[3].time := 3600.0, [44].log_data[3].valid := 1, [44].log_data[4].min := 0.48812497, [44].log_data[4].max := 0.841875, [44].log_data[4].total := 2360.5496, [44].log_data[4].time := 3600.0, [44].log_data[4].minminute := 1, [44].log_data[4].maxminute := 59, [44].log_data[4].valid := 1, [44].log_data[5].max := 7.12875, [44].log_data[5].total := 711.53986, [44].log_data[5].time := 3600.0, [44].log_data[5].minminute := 1, [44].log_data[5].valid := 1, [44].log_data[6].valid := 1, [44].log_data[7].valid := 1, [44].log_data[8].valid := 1, [44].log_data[9].valid := 1, [44].log_data[10].valid := 1, [44].log_data[11].valid := 1, [44].log_data[12].valid := 1, [44].log_data[13].valid := 1, [44].log_data[14].valid := 1, [44].log_data[15].valid := 1, [44].log_data[16].valid := 1, [44].log_data[17].valid := 1, [44].log_data[18].valid := 1, [44].log_data[19].valid := 1, [44].time.Year := 2022, [44].time.Month := 4, [44].time.Day := 28, [44].time.Hour := 13, [44].time.Minute := 59, [44].time.Second := 59, [44].time.DST_ON := 1, [45].log_data[0].min := 1.0, [45].log_data[0].max := 1.0, [45].log_data[0].total := 3599.999, [45].log_data[0].time := 3599.999, [45].log_data[0].valid := 1, [45].log_data[1].time := 3599.999, [45].log_data[1].valid := 1, [45].log_data[2].time := 3599.999, [45].log_data[2].valid := 1,
        [45].log_data[3].time := 3599.999, [45].log_data[3].valid := 1, [45].log_data[4].min := 0.84124994, [45].log_data[4].max := 0.995, [45].log_data[4].total := 3318.3955, [45].log_data[4].time := 3599.999, [45].log_data[4].maxminute := 59, [45].log_data[4].valid := 1, [45].log_data[5].time := 3599.999, [45].log_data[5].valid := 1, [45].log_data[6].valid := 1, [45].log_data[7].valid := 1, [45].log_data[8].valid := 1, [45].log_data[9].valid := 1, [45].log_data[10].valid := 1, [45].log_data[11].valid := 1, [45].log_data[12].valid := 1, [45].log_data[13].valid := 1, [45].log_data[14].valid := 1, [45].log_data[15].valid := 1, [45].log_data[16].valid := 1, [45].log_data[17].valid := 1, [45].log_data[18].valid := 1, [45].log_data[19].valid := 1, [45].time.Year := 2022, [45].time.Month := 4, [45].time.Day := 28, [45].time.Hour := 14, [45].time.Minute := 59, [45].time.Second := 59, [45].time.DST_ON := 1, [46].log_data[0].min := 1.0, [46].log_data[0].max := 1.0, [46].log_data[0].total := 3600.0, [46].log_data[0].time := 3600.0, [46].log_data[0].valid := 1, [46].log_data[1].time := 3600.0, [46].log_data[1].valid := 1, [46].log_data[2].max := 1.0, [46].log_data[2].total := 478.5, [46].log_data[2].time := 3600.0, [46].log_data[2].maxminute := 10, [46].log_data[2].valid := 1, [46].log_data[3].time := 3600.0, [46].log_data[3].valid := 1, [46].log_data[4].min := 0.48812497, [46].log_data[4].max := 1.0068749, [46].log_data[4].total := 2440.602, [46].log_data[4].time := 3600.0, [46].log_data[4].minminute := 18, [46].log_data[4].maxminute := 10, [46].log_data[4].valid := 1, [46].log_data[5].max := 7.2275, [46].log_data[5].total := 3392.0232, [46].log_data[5].time := 3600.0, [46].log_data[5].maxminute := 11, [46].log_data[5].valid := 1, [46].log_data[6].valid := 1, [46].log_data[7].valid := 1, [46].log_data[8].valid := 1,
        [46].log_data[9].valid := 1, [46].log_data[10].valid := 1, [46].log_data[11].valid := 1, [46].log_data[12].valid := 1, [46].log_data[13].valid := 1, [46].log_data[14].valid := 1, [46].log_data[15].valid := 1, [46].log_data[16].valid := 1, [46].log_data[17].valid := 1, [46].log_data[18].valid := 1, [46].log_data[19].valid := 1, [46].time.Year := 2022, [46].time.Month := 4, [46].time.Day := 28, [46].time.Hour := 15, [46].time.Minute := 59, [46].time.Second := 59, [46].time.DST_ON := 1, [47].log_data[0].min := 1.0, [47].log_data[0].max := 1.0, [47].log_data[0].total := 3600.0, [47].log_data[0].time := 3600.0, [47].log_data[0].valid := 1, [47].log_data[1].time := 3600.0, [47].log_data[1].valid := 1, [47].log_data[2].time := 3600.0, [47].log_data[2].valid := 1, [47].log_data[3].time := 3600.0, [47].log_data[3].valid := 1, [47].log_data[4].min := 0.6875, [47].log_data[4].max := 0.934375, [47].log_data[4].total := 3012.0981, [47].log_data[4].time := 3600.0, [47].log_data[4].maxminute := 59, [47].log_data[4].valid := 1, [47].log_data[5].time := 3600.0, [47].log_data[5].valid := 1, [47].log_data[6].valid := 1, [47].log_data[7].valid := 1, [47].log_data[8].valid := 1, [47].log_data[9].valid := 1, [47].log_data[10].valid := 1, [47].log_data[11].valid := 1, [47].log_data[12].valid := 1, [47].log_data[13].valid := 1, [47].log_data[14].valid := 1, [47].log_data[15].valid := 1, [47].log_data[16].valid := 1, [47].log_data[17].valid := 1, [47].log_data[18].valid := 1, [47].log_data[19].valid := 1, [47].time.Year := 2022, [47].time.Month := 4, [47].time.Day := 28, [47].time.Hour := 16, [47].time.Minute := 59, [47].time.Second := 59, [47].time.DST_ON := 1, [48].log_data[0].min := 1.0, [48].log_data[0].max := 1.0,
        [48].log_data[0].total := 3600.5, [48].log_data[0].time := 3600.5, [48].log_data[0].valid := 1, [48].log_data[1].max := 1.0, [48].log_data[1].total := 492.0, [48].log_data[1].time := 3600.5, [48].log_data[1].maxminute := 20, [48].log_data[1].valid := 1, [48].log_data[2].time := 3600.5, [48].log_data[2].valid := 1, [48].log_data[3].time := 3600.5, [48].log_data[3].valid := 1, [48].log_data[4].min := 0.48749998, [48].log_data[4].max := 1.00625, [48].log_data[4].total := 2704.1812, [48].log_data[4].time := 3600.5, [48].log_data[4].minminute := 28, [48].log_data[4].maxminute := 20, [48].log_data[4].valid := 1, [48].log_data[5].max := 7.1475, [48].log_data[5].total := 3460.189, [48].log_data[5].time := 3600.5, [48].log_data[5].maxminute := 20, [48].log_data[5].valid := 1, [48].log_data[6].valid := 1, [48].log_data[7].valid := 1, [48].log_data[8].valid := 1, [48].log_data[9].valid := 1, [48].log_data[10].valid := 1, [48].log_data[11].valid := 1, [48].log_data[12].valid := 1, [48].log_data[13].valid := 1, [48].log_data[14].valid := 1, [48].log_data[15].valid := 1, [48].log_data[16].valid := 1, [48].log_data[17].valid := 1, [48].log_data[18].valid := 1, [48].log_data[19].valid := 1, [48].time.Year := 2022, [48].time.Month := 4, [48].time.Day := 28, [48].time.Hour := 17, [48].time.Minute := 59, [48].time.Second := 59, [48].time.DST_ON := 1, [49].log_data[0].min := 1.0, [49].log_data[0].max := 1.0, [49].log_data[0].total := 3600.0, [49].log_data[0].time := 3600.0, [49].log_data[0].valid := 1, [49].log_data[1].time := 3600.0, [49].log_data[1].valid := 1, [49].log_data[2].time := 3600.0, [49].log_data[2].valid := 1, [49].log_data[3].time := 3600.0, [49].log_data[3].valid := 1, [49].log_data[4].min := 0.70375, [49].log_data[4].max := 0.94875, [49].log_data[4].total := 3048.5398, [49].log_data[4].time := 3600.0,
        [49].log_data[4].maxminute := 59, [49].log_data[4].valid := 1, [49].log_data[5].time := 3600.0, [49].log_data[5].valid := 1, [49].log_data[6].valid := 1, [49].log_data[7].valid := 1, [49].log_data[8].valid := 1, [49].log_data[9].valid := 1, [49].log_data[10].valid := 1, [49].log_data[11].valid := 1, [49].log_data[12].valid := 1, [49].log_data[13].valid := 1, [49].log_data[14].valid := 1, [49].log_data[15].valid := 1, [49].log_data[16].valid := 1, [49].log_data[17].valid := 1, [49].log_data[18].valid := 1, [49].log_data[19].valid := 1, [49].time.Year := 2022, [49].time.Month := 4, [49].time.Day := 28, [49].time.Hour := 18, [49].time.Minute := 59, [49].time.Second := 59, [49].time.DST_ON := 1, [50].log_data[0].min := 1.0, [50].log_data[0].max := 1.0, [50].log_data[0].total := 3600.0, [50].log_data[0].time := 3600.0, [50].log_data[0].valid := 1, [50].log_data[1].time := 3600.0, [50].log_data[1].valid := 1, [50].log_data[2].max := 1.0, [50].log_data[2].total := 501.0, [50].log_data[2].time := 3600.0, [50].log_data[2].maxminute := 17, [50].log_data[2].valid := 1, [50].log_data[3].time := 3600.0, [50].log_data[3].valid := 1, [50].log_data[4].min := 0.48749998, [50].log_data[4].max := 1.0068749, [50].log_data[4].total := 2793.4758, [50].log_data[4].time := 3600.0, [50].log_data[4].minminute := 25, [50].log_data[4].maxminute := 17, [50].log_data[4].valid := 1, [50].log_data[5].max := 7.21375, [50].log_data[5].total := 3548.544, [50].log_data[5].time := 3600.0, [50].log_data[5].maxminute := 18, [50].log_data[5].valid := 1, [50].log_data[6].valid := 1, [50].log_data[7].valid := 1, [50].log_data[8].valid := 1, [50].log_data[9].valid := 1, [50].log_data[10].valid := 1, [50].log_data[11].valid := 1, [50].log_data[12].valid := 1, [50].log_data[13].valid := 1, [50].log_data[14].valid := 1,
        [50].log_data[15].valid := 1, [50].log_data[16].valid := 1, [50].log_data[17].valid := 1, [50].log_data[18].valid := 1, [50].log_data[19].valid := 1, [50].time.Year := 2022, [50].time.Month := 4, [50].time.Day := 28, [50].time.Hour := 19, [50].time.Minute := 59, [50].time.Second := 59, [50].time.DST_ON := 1, [51].log_data[0].min := 1.0, [51].log_data[0].max := 1.0, [51].log_data[0].total := 3600.0, [51].log_data[0].time := 3600.0, [51].log_data[0].valid := 1, [51].log_data[1].max := 1.0, [51].log_data[1].total := 532.5, [51].log_data[1].time := 3600.0, [51].log_data[1].maxminute := 26, [51].log_data[1].valid := 1, [51].log_data[2].time := 3600.0, [51].log_data[2].valid := 1, [51].log_data[3].time := 3600.0, [51].log_data[3].valid := 1, [51].log_data[4].min := 0.48749998, [51].log_data[4].max := 1.00875, [51].log_data[4].total := 2873.0312, [51].log_data[4].time := 3600.0, [51].log_data[4].minminute := 35, [51].log_data[4].maxminute := 26, [51].log_data[4].valid := 1, [51].log_data[5].max := 7.1499996, [51].log_data[5].total := 3733.1885, [51].log_data[5].time := 3600.0, [51].log_data[5].maxminute := 27, [51].log_data[5].valid := 1, [51].log_data[6].valid := 1, [51].log_data[7].valid := 1, [51].log_data[8].valid := 1, [51].log_data[9].valid := 1, [51].log_data[10].valid := 1, [51].log_data[11].valid := 1, [51].log_data[12].valid := 1, [51].log_data[13].valid := 1, [51].log_data[14].valid := 1, [51].log_data[15].valid := 1, [51].log_data[16].valid := 1, [51].log_data[17].valid := 1, [51].log_data[18].valid := 1, [51].log_data[19].valid := 1, [51].time.Year := 2022, [51].time.Month := 4, [51].time.Day := 28, [51].time.Hour := 20, [51].time.Minute := 59, [51].time.Second := 59, [51].time.DST_ON := 1, [52].log_data[0].min := 1.0,
        [52].log_data[0].max := 1.0, [52].log_data[0].total := 3600.0, [52].log_data[0].time := 3600.0, [52].log_data[0].valid := 1, [52].log_data[1].time := 3600.0, [52].log_data[1].valid := 1, [52].log_data[2].max := 1.0, [52].log_data[2].total := 512.0, [52].log_data[2].time := 3600.0, [52].log_data[2].maxminute := 24, [52].log_data[2].valid := 1, [52].log_data[3].time := 3600.0, [52].log_data[3].valid := 1, [52].log_data[4].min := 0.48749998, [52].log_data[4].max := 1.0068749, [52].log_data[4].total := 2843.7546, [52].log_data[4].time := 3600.0, [52].log_data[4].minminute := 33, [52].log_data[4].maxminute := 24, [52].log_data[4].valid := 1, [52].log_data[5].max := 7.2250004, [52].log_data[5].total := 3628.2964, [52].log_data[5].time := 3600.0, [52].log_data[5].maxminute := 26, [52].log_data[5].valid := 1, [52].log_data[6].valid := 1, [52].log_data[7].valid := 1, [52].log_data[8].valid := 1, [52].log_data[9].valid := 1, [52].log_data[10].valid := 1, [52].log_data[11].valid := 1, [52].log_data[12].valid := 1, [52].log_data[13].valid := 1, [52].log_data[14].valid := 1, [52].log_data[15].valid := 1, [52].log_data[16].valid := 1, [52].log_data[17].valid := 1, [52].log_data[18].valid := 1, [52].log_data[19].valid := 1, [52].time.Year := 2022, [52].time.Month := 4, [52].time.Day := 28, [52].time.Hour := 21, [52].time.Minute := 59, [52].time.Second := 59, [52].time.DST_ON := 1, [53].log_data[0].min := 1.0, [53].log_data[0].max := 1.0, [53].log_data[0].total := 3600.0, [53].log_data[0].time := 3600.0, [53].log_data[0].valid := 1, [53].log_data[1].max := 1.0, [53].log_data[1].total := 506.0, [53].log_data[1].time := 3600.0, [53].log_data[1].maxminute := 28, [53].log_data[1].valid := 1, [53].log_data[2].time := 3600.0, [53].log_data[2].valid := 1, [53].log_data[3].time := 3600.0, [53].log_data[3].valid := 1,
        [53].log_data[4].min := 0.48812497, [53].log_data[4].max := 1.00875, [53].log_data[4].total := 2825.9617, [53].log_data[4].time := 3600.0, [53].log_data[4].minminute := 37, [53].log_data[4].maxminute := 28, [53].log_data[4].valid := 1, [53].log_data[5].max := 7.1949997, [53].log_data[5].total := 3580.4539, [53].log_data[5].time := 3600.0, [53].log_data[5].maxminute := 29, [53].log_data[5].valid := 1, [53].log_data[6].valid := 1, [53].log_data[7].valid := 1, [53].log_data[8].valid := 1, [53].log_data[9].valid := 1, [53].log_data[10].valid := 1, [53].log_data[11].valid := 1, [53].log_data[12].valid := 1, [53].log_data[13].valid := 1, [53].log_data[14].valid := 1, [53].log_data[15].valid := 1, [53].log_data[16].valid := 1, [53].log_data[17].valid := 1, [53].log_data[18].valid := 1, [53].log_data[19].valid := 1, [53].time.Year := 2022, [53].time.Month := 4, [53].time.Day := 28, [53].time.Hour := 22, [53].time.Minute := 59, [53].time.Second := 59, [53].time.DST_ON := 1, [54].log_data[0].min := 1.0, [54].log_data[0].max := 1.0, [54].log_data[0].total := 3600.0, [54].log_data[0].time := 3600.0, [54].log_data[0].valid := 1, [54].log_data[1].time := 3600.0, [54].log_data[1].valid := 1, [54].log_data[2].time := 3600.0, [54].log_data[2].valid := 1, [54].log_data[3].time := 3600.0, [54].log_data[3].valid := 1, [54].log_data[4].min := 0.674375, [54].log_data[4].max := 0.995, [54].log_data[4].total := 3131.7812, [54].log_data[4].time := 3600.0, [54].log_data[4].maxminute := 57, [54].log_data[4].valid := 1, [54].log_data[5].max := 0.0012500001, [54].log_data[5].total := 0.37750566, [54].log_data[5].time := 3600.0, [54].log_data[5].valid := 1, [54].log_data[6].valid := 1, [54].log_data[7].valid := 1, [54].log_data[8].valid := 1, [54].log_data[9].valid := 1, [54].log_data[10].valid := 1, [54].log_data[11].valid := 1,
        [54].log_data[12].valid := 1, [54].log_data[13].valid := 1, [54].log_data[14].valid := 1, [54].log_data[15].valid := 1, [54].log_data[16].valid := 1, [54].log_data[17].valid := 1, [54].log_data[18].valid := 1, [54].log_data[19].valid := 1, [54].time.Year := 2022, [54].time.Month := 4, [54].time.Day := 28, [54].time.Hour := 23, [54].time.Minute := 59, [54].time.Second := 59, [54].time.DST_ON := 1, [55].log_data[0].min := 1.0, [55].log_data[0].max := 1.0, [55].log_data[0].total := 3600.0, [55].log_data[0].time := 3600.0, [55].log_data[0].valid := 1, [55].log_data[1].time := 3600.0, [55].log_data[1].valid := 1, [55].log_data[2].max := 1.0, [55].log_data[2].total := 483.0, [55].log_data[2].time := 3600.0, [55].log_data[2].maxminute := 3, [55].log_data[2].valid := 1, [55].log_data[3].time := 3600.0, [55].log_data[3].valid := 1, [55].log_data[4].min := 0.48812497, [55].log_data[4].max := 1.005625, [55].log_data[4].total := 2437.0598, [55].log_data[4].time := 3600.0, [55].log_data[4].minminute := 12, [55].log_data[4].maxminute := 3, [55].log_data[4].valid := 1, [55].log_data[5].max := 7.2237496, [55].log_data[5].total := 3426.2332, [55].log_data[5].time := 3600.0, [55].log_data[5].maxminute := 4, [55].log_data[5].valid := 1, [55].log_data[6].valid := 1, [55].log_data[7].valid := 1, [55].log_data[8].valid := 1, [55].log_data[9].valid := 1, [55].log_data[10].valid := 1, [55].log_data[11].valid := 1, [55].log_data[12].valid := 1, [55].log_data[13].valid := 1, [55].log_data[14].valid := 1, [55].log_data[15].valid := 1, [55].log_data[16].valid := 1, [55].log_data[17].valid := 1, [55].log_data[18].valid := 1, [55].log_data[19].valid := 1, [55].time.Year := 2022, [55].time.Month := 4, [55].time.Day := 29, [55].time.Minute := 59, [55].time.Second := 59,
        [55].time.DST_ON := 1, [56].log_data[0].min := 1.0, [56].log_data[0].max := 1.0, [56].log_data[0].total := 3599.998, [56].log_data[0].time := 3599.998, [56].log_data[0].valid := 1, [56].log_data[1].time := 3599.998, [56].log_data[1].valid := 1, [56].log_data[2].time := 3599.998, [56].log_data[2].valid := 1, [56].log_data[3].time := 3599.998, [56].log_data[3].valid := 1, [56].log_data[4].min := 0.79499996, [56].log_data[4].max := 0.94875, [56].log_data[4].total := 3201.0476, [56].log_data[4].time := 3599.998, [56].log_data[4].maxminute := 58, [56].log_data[4].valid := 1, [56].log_data[5].max := 0.0025000002, [56].log_data[5].total := 1.9639266, [56].log_data[5].time := 3599.998, [56].log_data[5].maxminute := 22, [56].log_data[5].valid := 1, [56].log_data[6].valid := 1, [56].log_data[7].valid := 1, [56].log_data[8].valid := 1, [56].log_data[9].valid := 1, [56].log_data[10].valid := 1, [56].log_data[11].valid := 1, [56].log_data[12].valid := 1, [56].log_data[13].valid := 1, [56].log_data[14].valid := 1, [56].log_data[15].valid := 1, [56].log_data[16].valid := 1, [56].log_data[17].valid := 1, [56].log_data[18].valid := 1, [56].log_data[19].valid := 1, [56].time.Year := 2022, [56].time.Month := 4, [56].time.Day := 29, [56].time.Hour := 1, [56].time.Minute := 59, [56].time.Second := 59, [56].time.DST_ON := 1, [57].log_data[0].min := 1.0, [57].log_data[0].max := 1.0, [57].log_data[0].total := 3600.0, [57].log_data[0].time := 3600.0, [57].log_data[0].valid := 1, [57].log_data[1].max := 1.0, [57].log_data[1].total := 475.0, [57].log_data[1].time := 3600.0, [57].log_data[1].maxminute := 45, [57].log_data[1].valid := 1, [57].log_data[2].time := 3600.0, [57].log_data[2].valid := 1, [57].log_data[3].time := 3600.0, [57].log_data[3].valid := 1, [57].log_data[4].min := 0.48812497, [57].log_data[4].max := 1.0081251,
        [57].log_data[4].total := 3232.466, [57].log_data[4].time := 3600.0, [57].log_data[4].minminute := 53, [57].log_data[4].maxminute := 45, [57].log_data[4].valid := 1, [57].log_data[5].max := 7.1525, [57].log_data[5].total := 3336.2666, [57].log_data[5].time := 3600.0, [57].log_data[5].maxminute := 45, [57].log_data[5].valid := 1, [57].log_data[6].valid := 1, [57].log_data[7].valid := 1, [57].log_data[8].valid := 1, [57].log_data[9].valid := 1, [57].log_data[10].valid := 1, [57].log_data[11].valid := 1, [57].log_data[12].valid := 1, [57].log_data[13].valid := 1, [57].log_data[14].valid := 1, [57].log_data[15].valid := 1, [57].log_data[16].valid := 1, [57].log_data[17].valid := 1, [57].log_data[18].valid := 1, [57].log_data[19].valid := 1, [57].time.Year := 2022, [57].time.Month := 4, [57].time.Day := 29, [57].time.Hour := 2, [57].time.Minute := 59, [57].time.Second := 59, [57].time.DST_ON := 1, [58].log_data[0].min := 1.0, [58].log_data[0].max := 1.0, [58].log_data[0].total := 3600.0, [58].log_data[0].time := 3600.0, [58].log_data[0].valid := 1, [58].log_data[1].time := 3600.0, [58].log_data[1].valid := 1, [58].log_data[2].time := 3600.0, [58].log_data[2].valid := 1, [58].log_data[3].time := 3600.0, [58].log_data[3].valid := 1, [58].log_data[4].min := 0.50374997, [58].log_data[4].max := 0.62687504, [58].log_data[4].total := 2036.3567, [58].log_data[4].time := 3600.0, [58].log_data[4].maxminute := 58, [58].log_data[4].valid := 1, [58].log_data[5].max := 0.0025000002, [58].log_data[5].total := 2.41244, [58].log_data[5].time := 3600.0, [58].log_data[5].maxminute := 16, [58].log_data[5].valid := 1, [58].log_data[6].valid := 1, [58].log_data[7].valid := 1, [58].log_data[8].valid := 1, [58].log_data[9].valid := 1, [58].log_data[10].valid := 1, [58].log_data[11].valid := 1, [58].log_data[12].valid := 1,
        [58].log_data[13].valid := 1, [58].log_data[14].valid := 1, [58].log_data[15].valid := 1, [58].log_data[16].valid := 1, [58].log_data[17].valid := 1, [58].log_data[18].valid := 1, [58].log_data[19].valid := 1, [58].time.Year := 2022, [58].time.Month := 4, [58].time.Day := 29, [58].time.Hour := 3, [58].time.Minute := 59, [58].time.Second := 59, [58].time.DST_ON := 1, [59].log_data[0].min := 1.0, [59].log_data[0].max := 1.0, [59].log_data[0].total := 3600.0, [59].log_data[0].time := 3600.0, [59].log_data[0].valid := 1, [59].log_data[1].time := 3600.0, [59].log_data[1].valid := 1, [59].log_data[2].time := 3600.0, [59].log_data[2].valid := 1, [59].log_data[3].time := 3600.0, [59].log_data[3].valid := 1, [59].log_data[4].min := 0.62624997, [59].log_data[4].max := 0.71875, [59].log_data[4].total := 2410.382, [59].log_data[4].time := 3600.0, [59].log_data[4].maxminute := 58, [59].log_data[4].valid := 1, [59].log_data[5].max := 0.0012500001, [59].log_data[5].total := 3.0441375, [59].log_data[5].time := 3600.0, [59].log_data[5].valid := 1, [59].log_data[6].valid := 1, [59].log_data[7].valid := 1, [59].log_data[8].valid := 1, [59].log_data[9].valid := 1, [59].log_data[10].valid := 1, [59].log_data[11].valid := 1, [59].log_data[12].valid := 1, [59].log_data[13].valid := 1, [59].log_data[14].valid := 1, [59].log_data[15].valid := 1, [59].log_data[16].valid := 1, [59].log_data[17].valid := 1, [59].log_data[18].valid := 1, [59].log_data[19].valid := 1, [59].time.Year := 2022, [59].time.Month := 4, [59].time.Day := 29, [59].time.Hour := 4, [59].time.Minute := 59, [59].time.Second := 59, [59].time.DST_ON := 1, [60].log_data[0].min := 1.0, [60].log_data[0].max := 1.0, [60].log_data[0].total := 3600.0, [60].log_data[0].time := 3600.0,
        [60].log_data[0].valid := 1, [60].log_data[1].time := 3600.0, [60].log_data[1].valid := 1, [60].log_data[2].time := 3600.0, [60].log_data[2].valid := 1, [60].log_data[3].time := 3600.0, [60].log_data[3].valid := 1, [60].log_data[4].min := 0.71812505, [60].log_data[4].max := 0.81125, [60].log_data[4].total := 2747.4373, [60].log_data[4].time := 3600.0, [60].log_data[4].maxminute := 59, [60].log_data[4].valid := 1, [60].log_data[5].max := 0.0025000002, [60].log_data[5].total := 3.147283, [60].log_data[5].time := 3600.0, [60].log_data[5].maxminute := 49, [60].log_data[5].valid := 1, [60].log_data[6].valid := 1, [60].log_data[7].valid := 1, [60].log_data[8].valid := 1, [60].log_data[9].valid := 1, [60].log_data[10].valid := 1, [60].log_data[11].valid := 1, [60].log_data[12].valid := 1, [60].log_data[13].valid := 1, [60].log_data[14].valid := 1, [60].log_data[15].valid := 1, [60].log_data[16].valid := 1, [60].log_data[17].valid := 1, [60].log_data[18].valid := 1, [60].log_data[19].valid := 1, [60].time.Year := 2022, [60].time.Month := 4, [60].time.Day := 29, [60].time.Hour := 5, [60].time.Minute := 59, [60].time.Second := 59, [60].time.DST_ON := 1, [61].log_data[0].min := 1.0, [61].log_data[0].max := 1.0, [61].log_data[0].total := 3599.999, [61].log_data[0].time := 3599.999, [61].log_data[0].valid := 1, [61].log_data[1].time := 3599.999, [61].log_data[1].valid := 1, [61].log_data[2].time := 3599.999, [61].log_data[2].valid := 1, [61].log_data[3].time := 3599.999, [61].log_data[3].valid := 1, [61].log_data[4].min := 0.81, [61].log_data[4].max := 0.90312505, [61].log_data[4].total := 3102.4812, [61].log_data[4].time := 3599.999, [61].log_data[4].maxminute := 57, [61].log_data[4].valid := 1, [61].log_data[5].max := 0.0012500001, [61].log_data[5].total := 3.1197772, [61].log_data[5].time := 3599.999, [61].log_data[5].valid := 1,
        [61].log_data[6].valid := 1, [61].log_data[7].valid := 1, [61].log_data[8].valid := 1, [61].log_data[9].valid := 1, [61].log_data[10].valid := 1, [61].log_data[11].valid := 1, [61].log_data[12].valid := 1, [61].log_data[13].valid := 1, [61].log_data[14].valid := 1, [61].log_data[15].valid := 1, [61].log_data[16].valid := 1, [61].log_data[17].valid := 1, [61].log_data[18].valid := 1, [61].log_data[19].valid := 1, [61].time.Year := 2022, [61].time.Month := 4, [61].time.Day := 29, [61].time.Hour := 6, [61].time.Minute := 59, [61].time.Second := 59, [61].time.DST_ON := 1, [62].log_data[0].min := 1.0, [62].log_data[0].max := 1.0, [62].log_data[0].total := 3599.999, [62].log_data[0].time := 3599.999, [62].log_data[0].valid := 1, [62].log_data[1].time := 3599.999, [62].log_data[1].valid := 1, [62].log_data[2].time := 3599.999, [62].log_data[2].valid := 1, [62].log_data[3].time := 3599.999, [62].log_data[3].valid := 1, [62].log_data[4].min := 0.9024999, [62].log_data[4].max := 0.98, [62].log_data[4].total := 3353.119, [62].log_data[4].time := 3599.999, [62].log_data[4].maxminute := 59, [62].log_data[4].valid := 1, [62].log_data[5].max := 0.0025000002, [62].log_data[5].total := 2.1877053, [62].log_data[5].time := 3599.999, [62].log_data[5].maxminute := 15, [62].log_data[5].valid := 1, [62].log_data[6].valid := 1, [62].log_data[7].valid := 1, [62].log_data[8].valid := 1, [62].log_data[9].valid := 1, [62].log_data[10].valid := 1, [62].log_data[11].valid := 1, [62].log_data[12].valid := 1, [62].log_data[13].valid := 1, [62].log_data[14].valid := 1, [62].log_data[15].valid := 1, [62].log_data[16].valid := 1, [62].log_data[17].valid := 1, [62].log_data[18].valid := 1, [62].log_data[19].valid := 1, [62].time.Year := 2022, [62].time.Month := 4, [62].time.Day := 29,
        [62].time.Hour := 7, [62].time.Minute := 59, [62].time.Second := 59, [62].time.DST_ON := 1, [63].log_data[0].min := 1.0, [63].log_data[0].max := 1.0, [63].log_data[0].total := 3600.0, [63].log_data[0].time := 3600.0, [63].log_data[0].valid := 1, [63].log_data[1].time := 3600.0, [63].log_data[1].valid := 1, [63].log_data[2].max := 1.0, [63].log_data[2].total := 497.0, [63].log_data[2].time := 3600.0, [63].log_data[2].maxminute := 14, [63].log_data[2].valid := 1, [63].log_data[3].time := 3600.0, [63].log_data[3].valid := 1, [63].log_data[4].min := 0.48812497, [63].log_data[4].max := 1.005, [63].log_data[4].total := 2806.6924, [63].log_data[4].time := 3600.0, [63].log_data[4].minminute := 23, [63].log_data[4].maxminute := 14, [63].log_data[4].valid := 1, [63].log_data[5].max := 7.26, [63].log_data[5].total := 3541.7246, [63].log_data[5].time := 3600.0, [63].log_data[5].maxminute := 16, [63].log_data[5].valid := 1, [63].log_data[6].valid := 1, [63].log_data[7].valid := 1, [63].log_data[8].valid := 1, [63].log_data[9].valid := 1, [63].log_data[10].valid := 1, [63].log_data[11].valid := 1, [63].log_data[12].valid := 1, [63].log_data[13].valid := 1, [63].log_data[14].valid := 1, [63].log_data[15].valid := 1, [63].log_data[16].valid := 1, [63].log_data[17].valid := 1, [63].log_data[18].valid := 1, [63].log_data[19].valid := 1, [63].time.Year := 2022, [63].time.Month := 4, [63].time.Day := 29, [63].time.Hour := 8, [63].time.Minute := 59, [63].time.Second := 59, [63].time.DST_ON := 1, [64].log_data[0].min := 1.0, [64].log_data[0].max := 1.0, [64].log_data[0].total := 3599.999, [64].log_data[0].time := 3599.999, [64].log_data[0].valid := 1, [64].log_data[1].max := 1.0, [64].log_data[1].total := 492.5, [64].log_data[1].time := 3599.999, [64].log_data[1].maxminute := 34,
